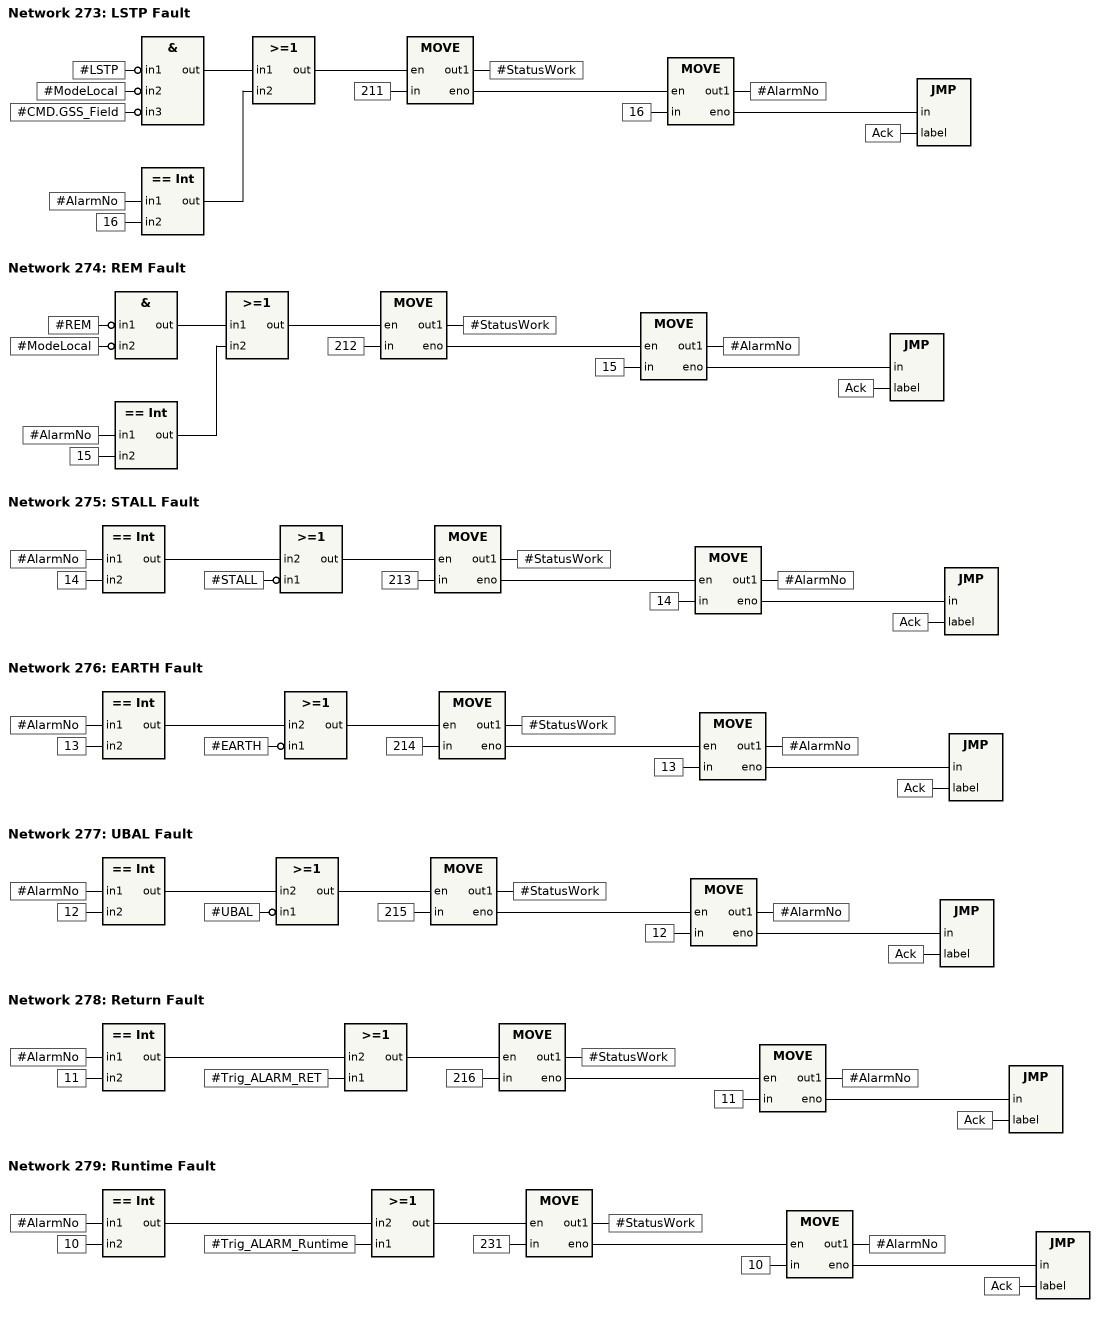
   // ENO of a box is taken as its EN; it also drops when the box reports an error
   #_w1 := (NOT #LSTP AND NOT #ModeLocal AND NOT #CMD.GSS_Field) OR (#AlarmNo = 16);
   IF #_w1 THEN
       #StatusWork := 211;
       #AlarmNo := 16;
       GOTO Ack;
   END_IF;
END_REGION

REGION Network 274: REM Fault
   // ENO of a box is taken as its EN; it also drops when the box reports an error
   #_w1 := (NOT #REM AND NOT #ModeLocal) OR (#AlarmNo = 15);
   IF #_w1 THEN
       #StatusWork := 212;
       #AlarmNo := 15;
       GOTO Ack;
   END_IF;
END_REGION

REGION Network 275: STALL Fault
   // ENO of a box is taken as its EN; it also drops when the box reports an error
   #_w1 := (#AlarmNo = 14) OR NOT #STALL;
   IF #_w1 THEN
       #StatusWork := 213;
       #AlarmNo := 14;
       GOTO Ack;
   END_IF;
END_REGION

REGION Network 276: EARTH Fault
   // ENO of a box is taken as its EN; it also drops when the box reports an error
   #_w1 := (#AlarmNo = 13) OR NOT #EARTH;
   IF #_w1 THEN
       #StatusWork := 214;
       #AlarmNo := 13;
       GOTO Ack;
   END_IF;
END_REGION

REGION Network 277: UBAL Fault
   // ENO of a box is taken as its EN; it also drops when the box reports an error
   #_w1 := (#AlarmNo = 12) OR NOT #UBAL;
   IF #_w1 THEN
       #StatusWork := 215;
       #AlarmNo := 12;
       GOTO Ack;
   END_IF;
END_REGION

REGION Network 278: Return Fault
   // ENO of a box is taken as its EN; it also drops when the box reports an error
   #_w1 := (#AlarmNo = 11) OR #Trig_ALARM_RET;
   IF #_w1 THEN
       #StatusWork := 216;
       #AlarmNo := 11;
       GOTO Ack;
   END_IF;
END_REGION

REGION Network 279: Runtime Fault
   // ENO of a box is taken as its EN; it also drops when the box reports an error
   #_w1 := (#AlarmNo = 10) OR #Trig_ALARM_Runtime;
   IF #_w1 THEN
       #StatusWork := 231;
       #AlarmNo := 10;
       GOTO Ack;
   END_IF;
END_REGION

REGION Network 280: Alarm Switch 1
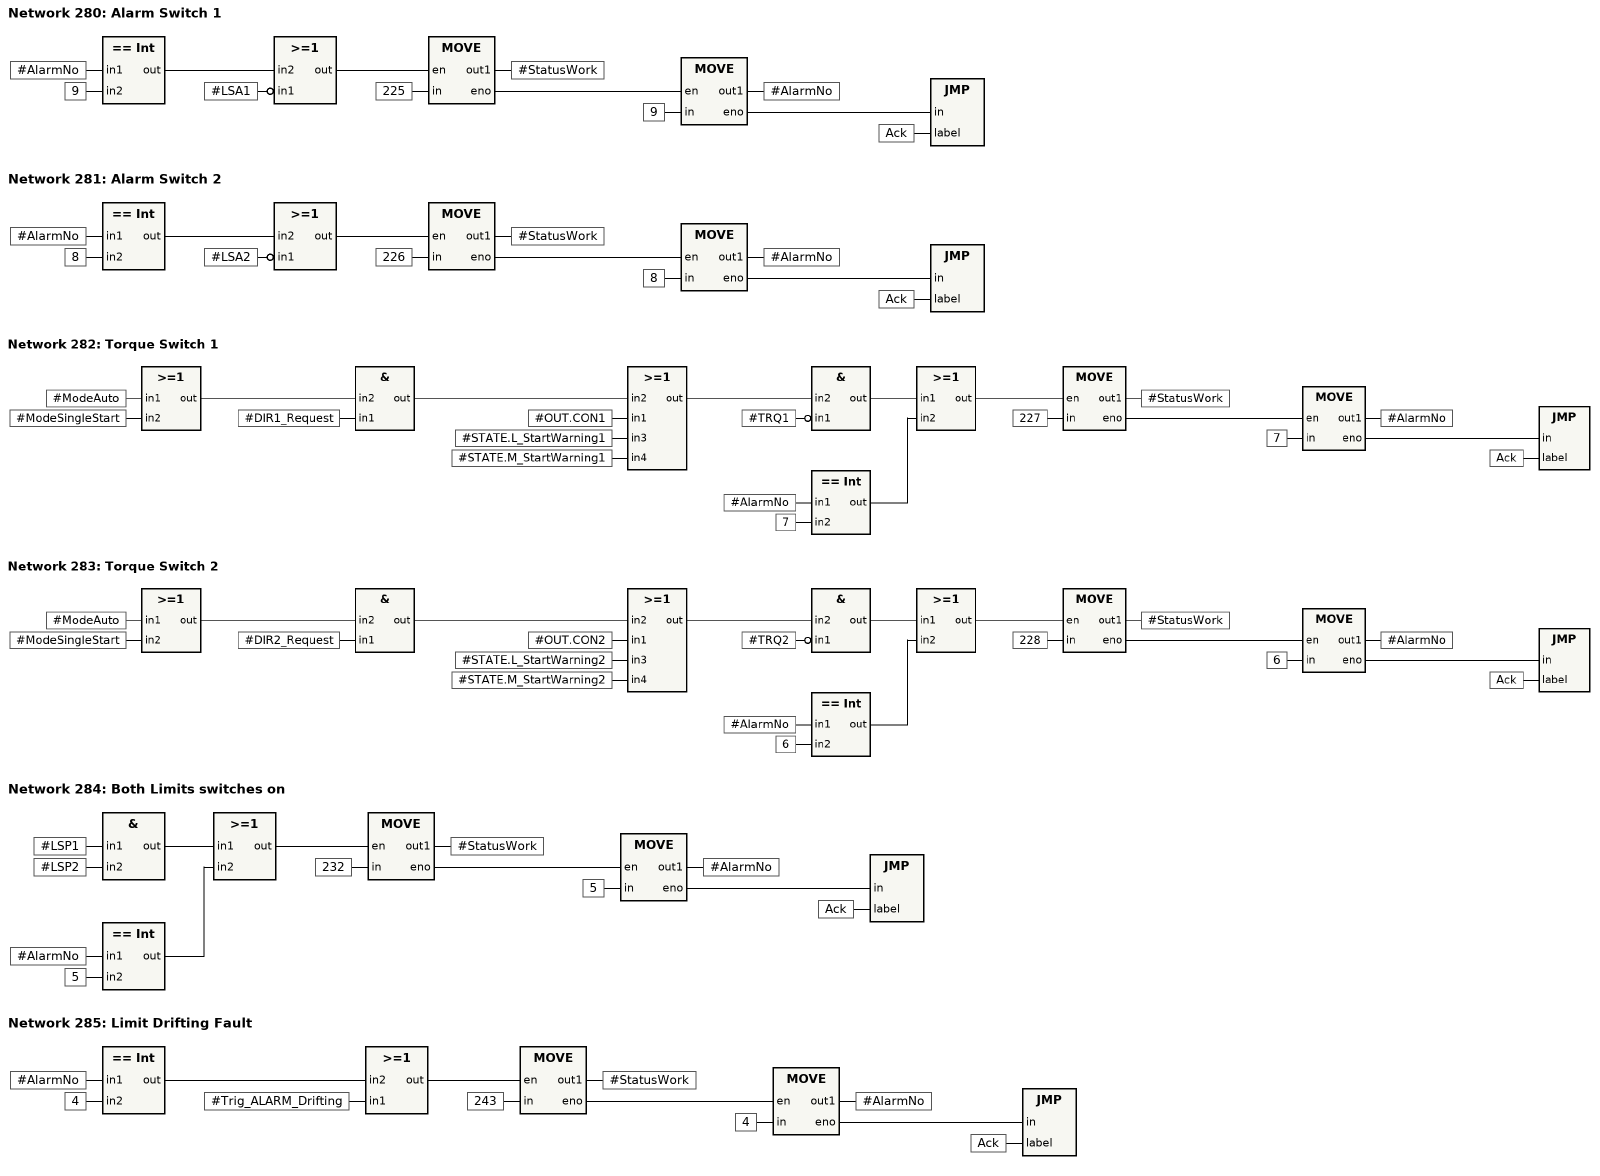
   // ENO of a box is taken as its EN; it also drops when the box reports an error
   #_w1 := (#AlarmNo = 9) OR NOT #LSA1;
   IF #_w1 THEN
       #StatusWork := 225;
       #AlarmNo := 9;
       GOTO Ack;
   END_IF;
END_REGION

REGION Network 281: Alarm Switch 2
   // ENO of a box is taken as its EN; it also drops when the box reports an error
   #_w1 := (#AlarmNo = 8) OR NOT #LSA2;
   IF #_w1 THEN
       #StatusWork := 226;
       #AlarmNo := 8;
       GOTO Ack;
   END_IF;
END_REGION

REGION Network 282: Torque Switch 1
   // Build 006 - 28 Jan 2020 (EXTBOB) : Torque fault considered in Local & Manual start
   // ENO of a box is taken as its EN; it also drops when the box reports an error
   #_w1 := ((((#ModeAuto OR #ModeSingleStart) AND #DIR1_Request) OR #OUT.CON1 OR #STATE.L_StartWarning1 OR #STATE.M_StartWarning1) AND NOT #TRQ1) OR (#AlarmNo = 7);
   IF #_w1 THEN
       #StatusWork := 227;
       #AlarmNo := 7;
       GOTO Ack;
   END_IF;
END_REGION

REGION Network 283: Torque Switch 2
   // Build 006 - 28 Jan 2020 (EXTBOB) : Torque fault considered in Local & Manual start
   // ENO of a box is taken as its EN; it also drops when the box reports an error
   #_w1 := ((((#ModeAuto OR #ModeSingleStart) AND #DIR2_Request) OR #OUT.CON2 OR #STATE.L_StartWarning2 OR #STATE.M_StartWarning2) AND NOT #TRQ2) OR (#AlarmNo = 6);
   IF #_w1 THEN
       #StatusWork := 228;
       #AlarmNo := 6;
       GOTO Ack;
   END_IF;
END_REGION

REGION Network 284: Both Limits switches on
   // ENO of a box is taken as its EN; it also drops when the box reports an error
   #_w1 := (#LSP1 AND #LSP2) OR (#AlarmNo = 5);
   IF #_w1 THEN
       #StatusWork := 232;
       #AlarmNo := 5;
       GOTO Ack;
   END_IF;
END_REGION

REGION Network 285: Limit Drifting Fault
   // ENO of a box is taken as its EN; it also drops when the box reports an error
   #_w1 := (#AlarmNo = 4) OR #Trig_ALARM_Drifting;
   IF #_w1 THEN
       #StatusWork := 243;
       #AlarmNo := 4;
       GOTO Ack;
   END_IF;
END_REGION

REGION Network 286: Analog pos Fault
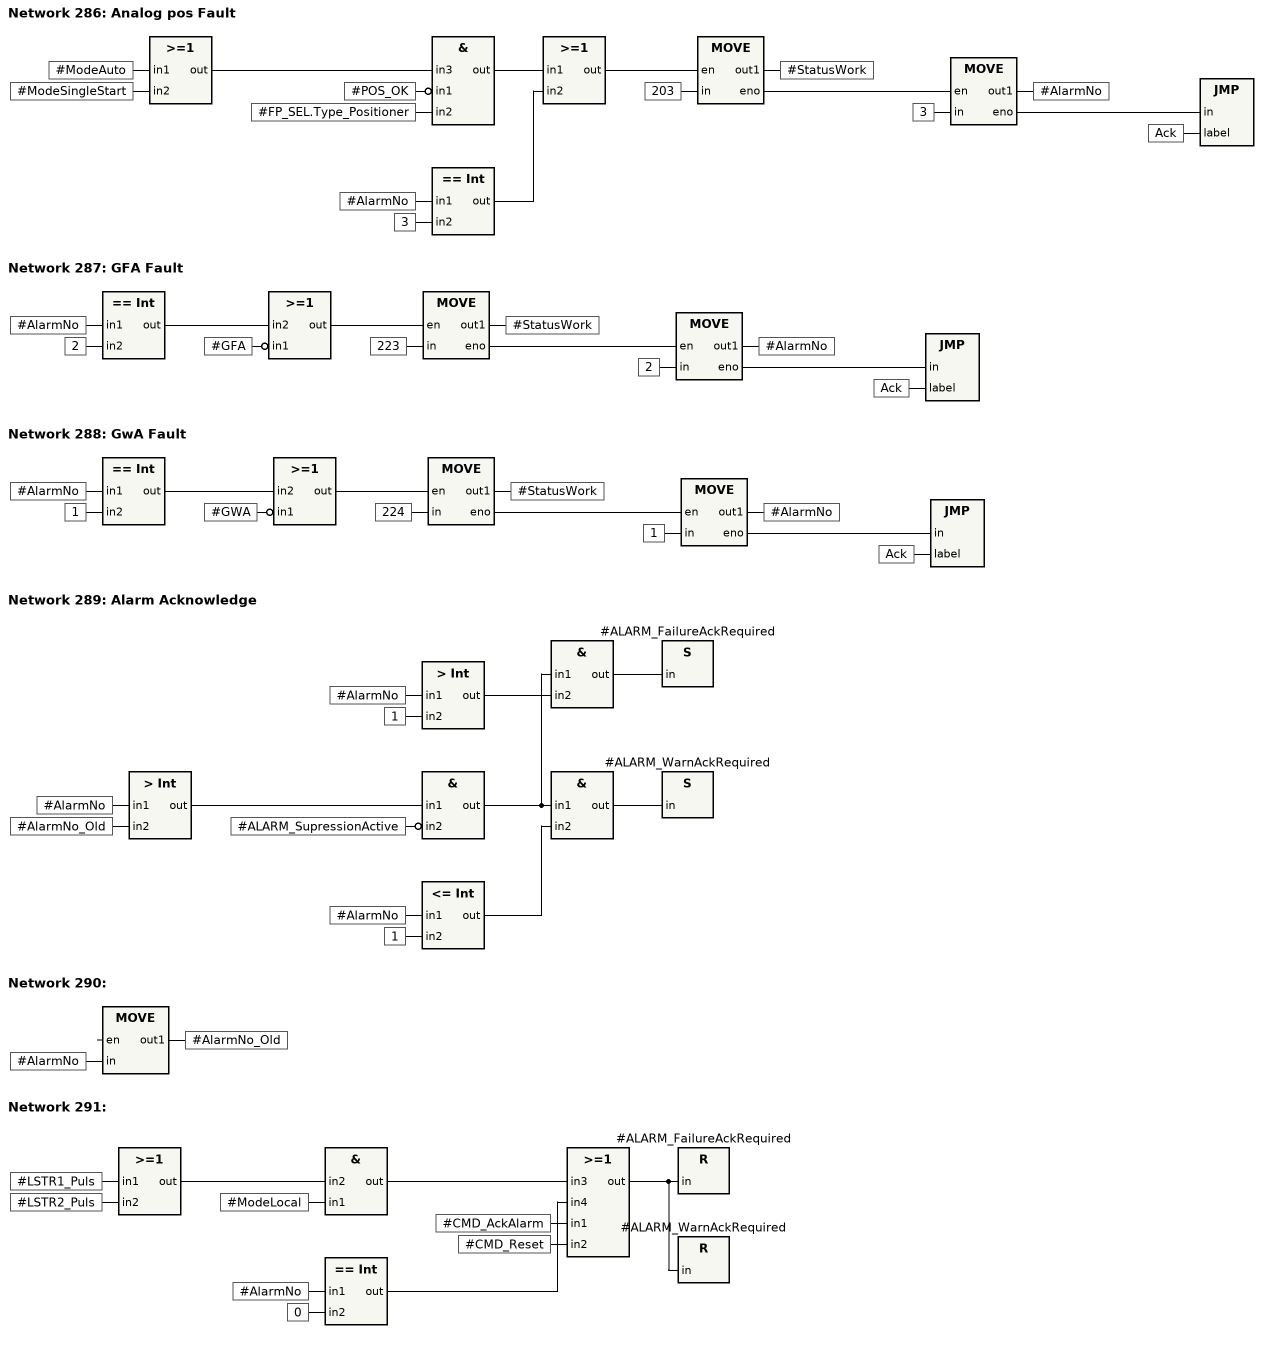
   // ENO of a box is taken as its EN; it also drops when the box reports an error
   #_w1 := ((#ModeAuto OR #ModeSingleStart) AND NOT #POS_OK AND #FP_SEL.Type_Positioner) OR (#AlarmNo = 3);
   IF #_w1 THEN
       #StatusWork := 203;
       #AlarmNo := 3;
       GOTO Ack;
   END_IF;
END_REGION

REGION Network 287: GFA Fault
   // ENO of a box is taken as its EN; it also drops when the box reports an error
   #_w1 := (#AlarmNo = 2) OR NOT #GFA;
   IF #_w1 THEN
       #StatusWork := 223;
       #AlarmNo := 2;
       GOTO Ack;
   END_IF;
END_REGION

REGION Network 288: GwA Fault
   // ENO of a box is taken as its EN; it also drops when the box reports an error
   #_w1 := (#AlarmNo = 1) OR NOT #GWA;
   IF #_w1 THEN
       #StatusWork := 224;
       #AlarmNo := 1;
       GOTO Ack;
   END_IF;
END_REGION

REGION Network 289: Alarm Acknowledge
   Ack:
   #_w1 := (#AlarmNo > #AlarmNo_Old) AND NOT #ALARM_SupressionActive;
   IF #_w1 AND (#AlarmNo > 1) THEN #ALARM_FailureAckRequired := TRUE; END_IF;
   IF #_w1 AND (#AlarmNo <= 1) THEN #ALARM_WarnAckRequired := TRUE; END_IF;
END_REGION

REGION Network 290
   #AlarmNo_Old := #AlarmNo;
END_REGION

REGION Network 291
   IF ((#LSTR1_Puls OR #LSTR2_Puls) AND #ModeLocal) OR (#AlarmNo = 0) OR #CMD_AckAlarm OR #CMD_Reset THEN
       #ALARM_FailureAckRequired := FALSE;
       #ALARM_WarnAckRequired := FALSE;
   END_IF;
END_REGION

REGION Network 292
   // Build 006 - 28 Jan 2020 (EXTBOB) : AlarmNo 6 and 7 Added to prevent Auto ack in torque falut
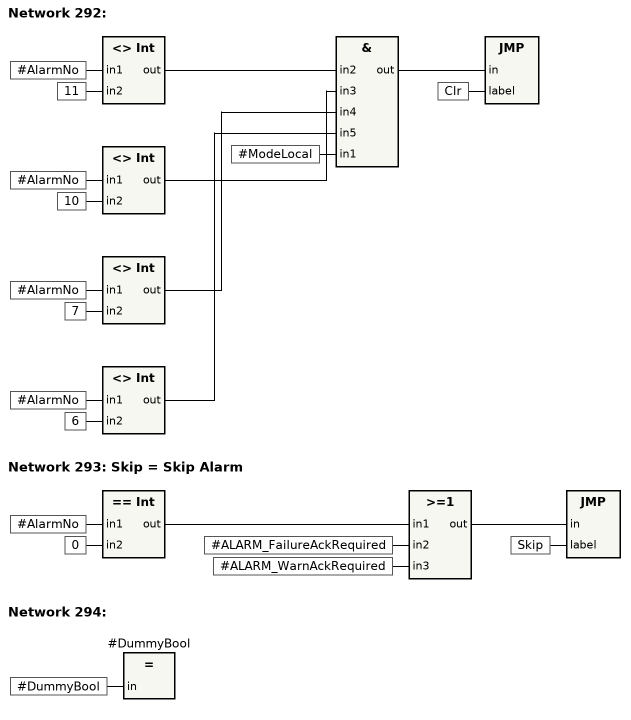
   IF (#AlarmNo <> 11) AND (#AlarmNo <> 10) AND (#AlarmNo <> 7) AND (#AlarmNo <> 6) AND #ModeLocal THEN
       GOTO Clr;
   END_IF;
END_REGION

REGION Network 293: Skip = Skip Alarm
   IF (#AlarmNo = 0) OR #ALARM_FailureAckRequired OR #ALARM_WarnAckRequired THEN GOTO Skip; END_IF;
END_REGION

REGION Network 294
   Clr:
   #DummyBool := #DummyBool;
END_REGION

REGION Network 295
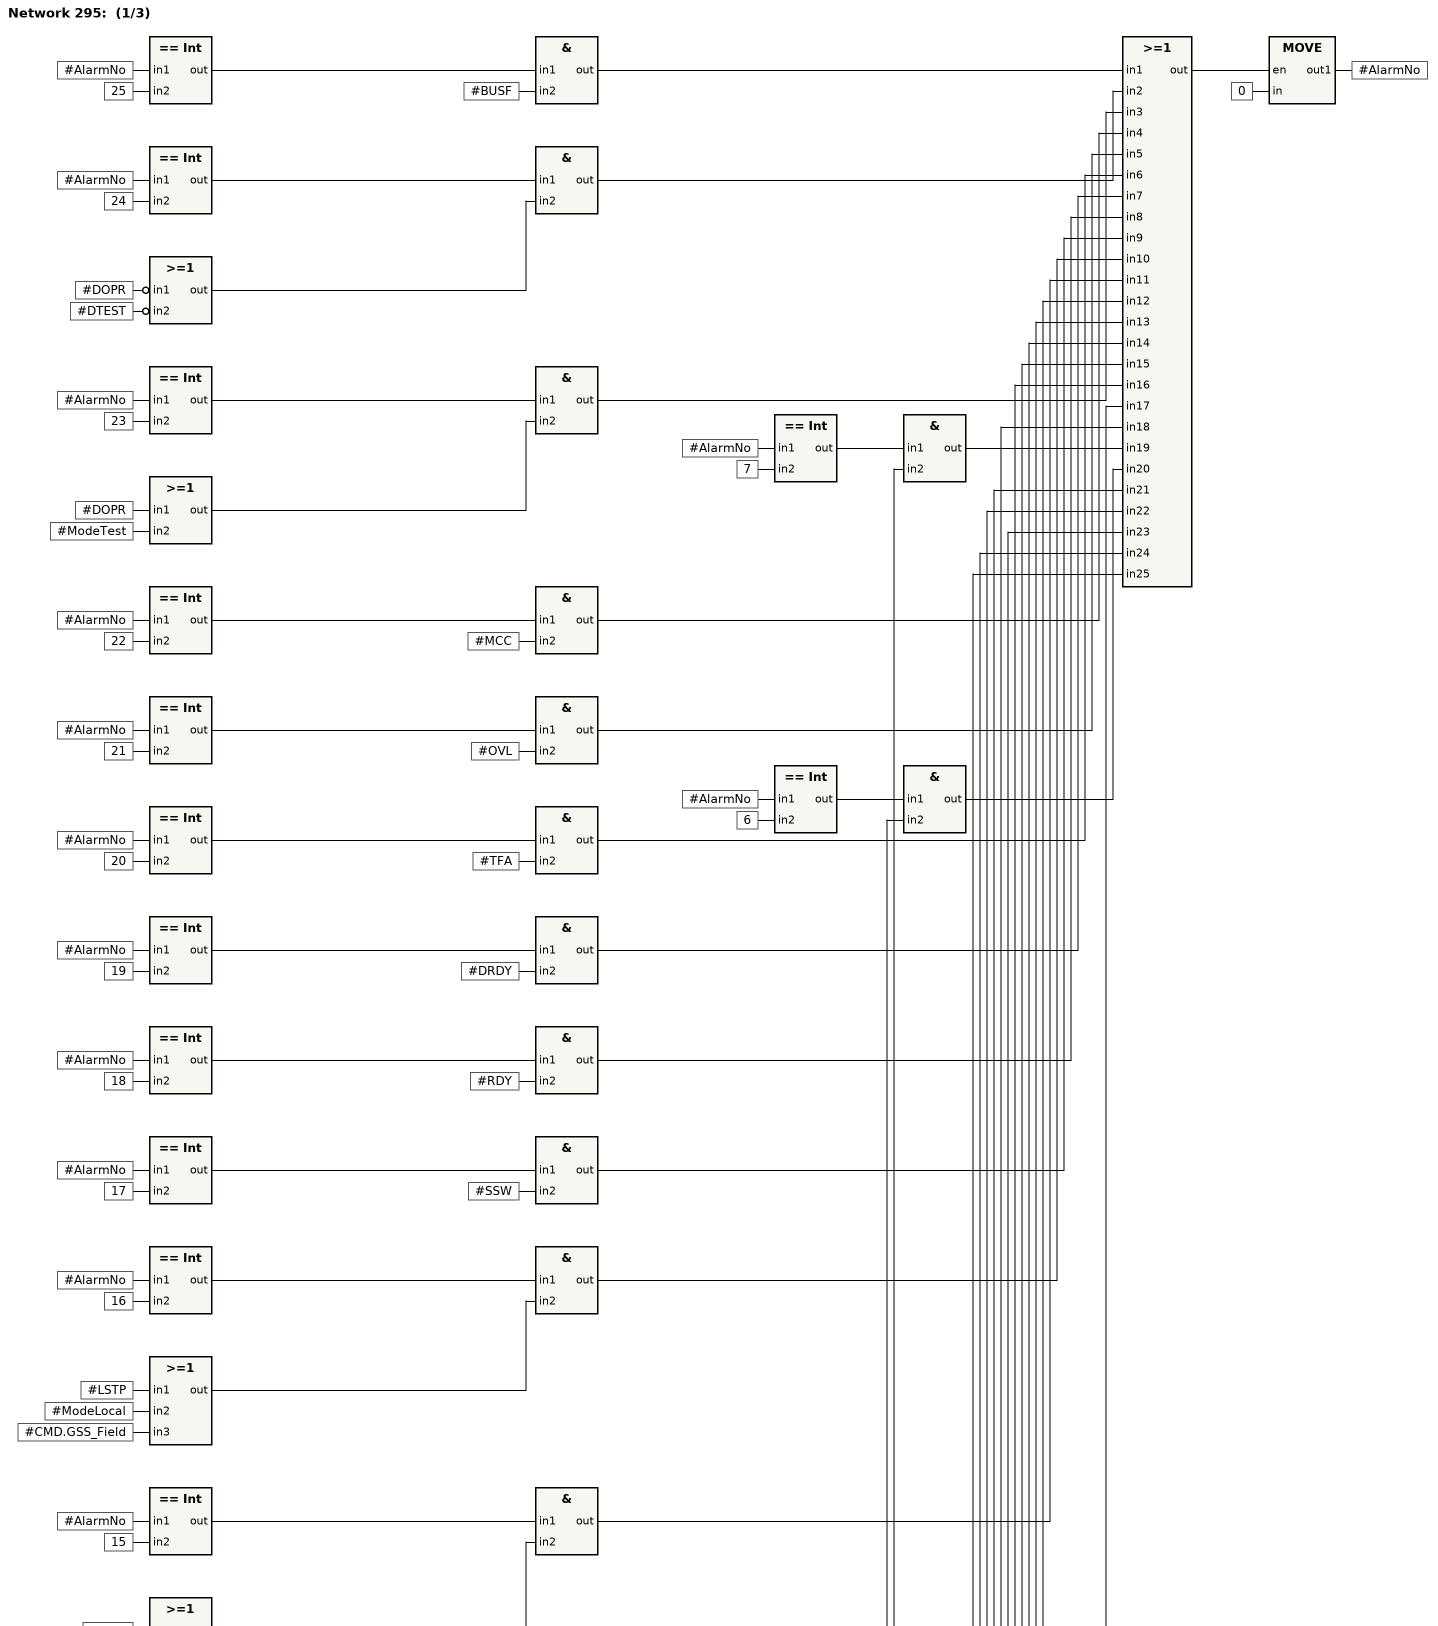
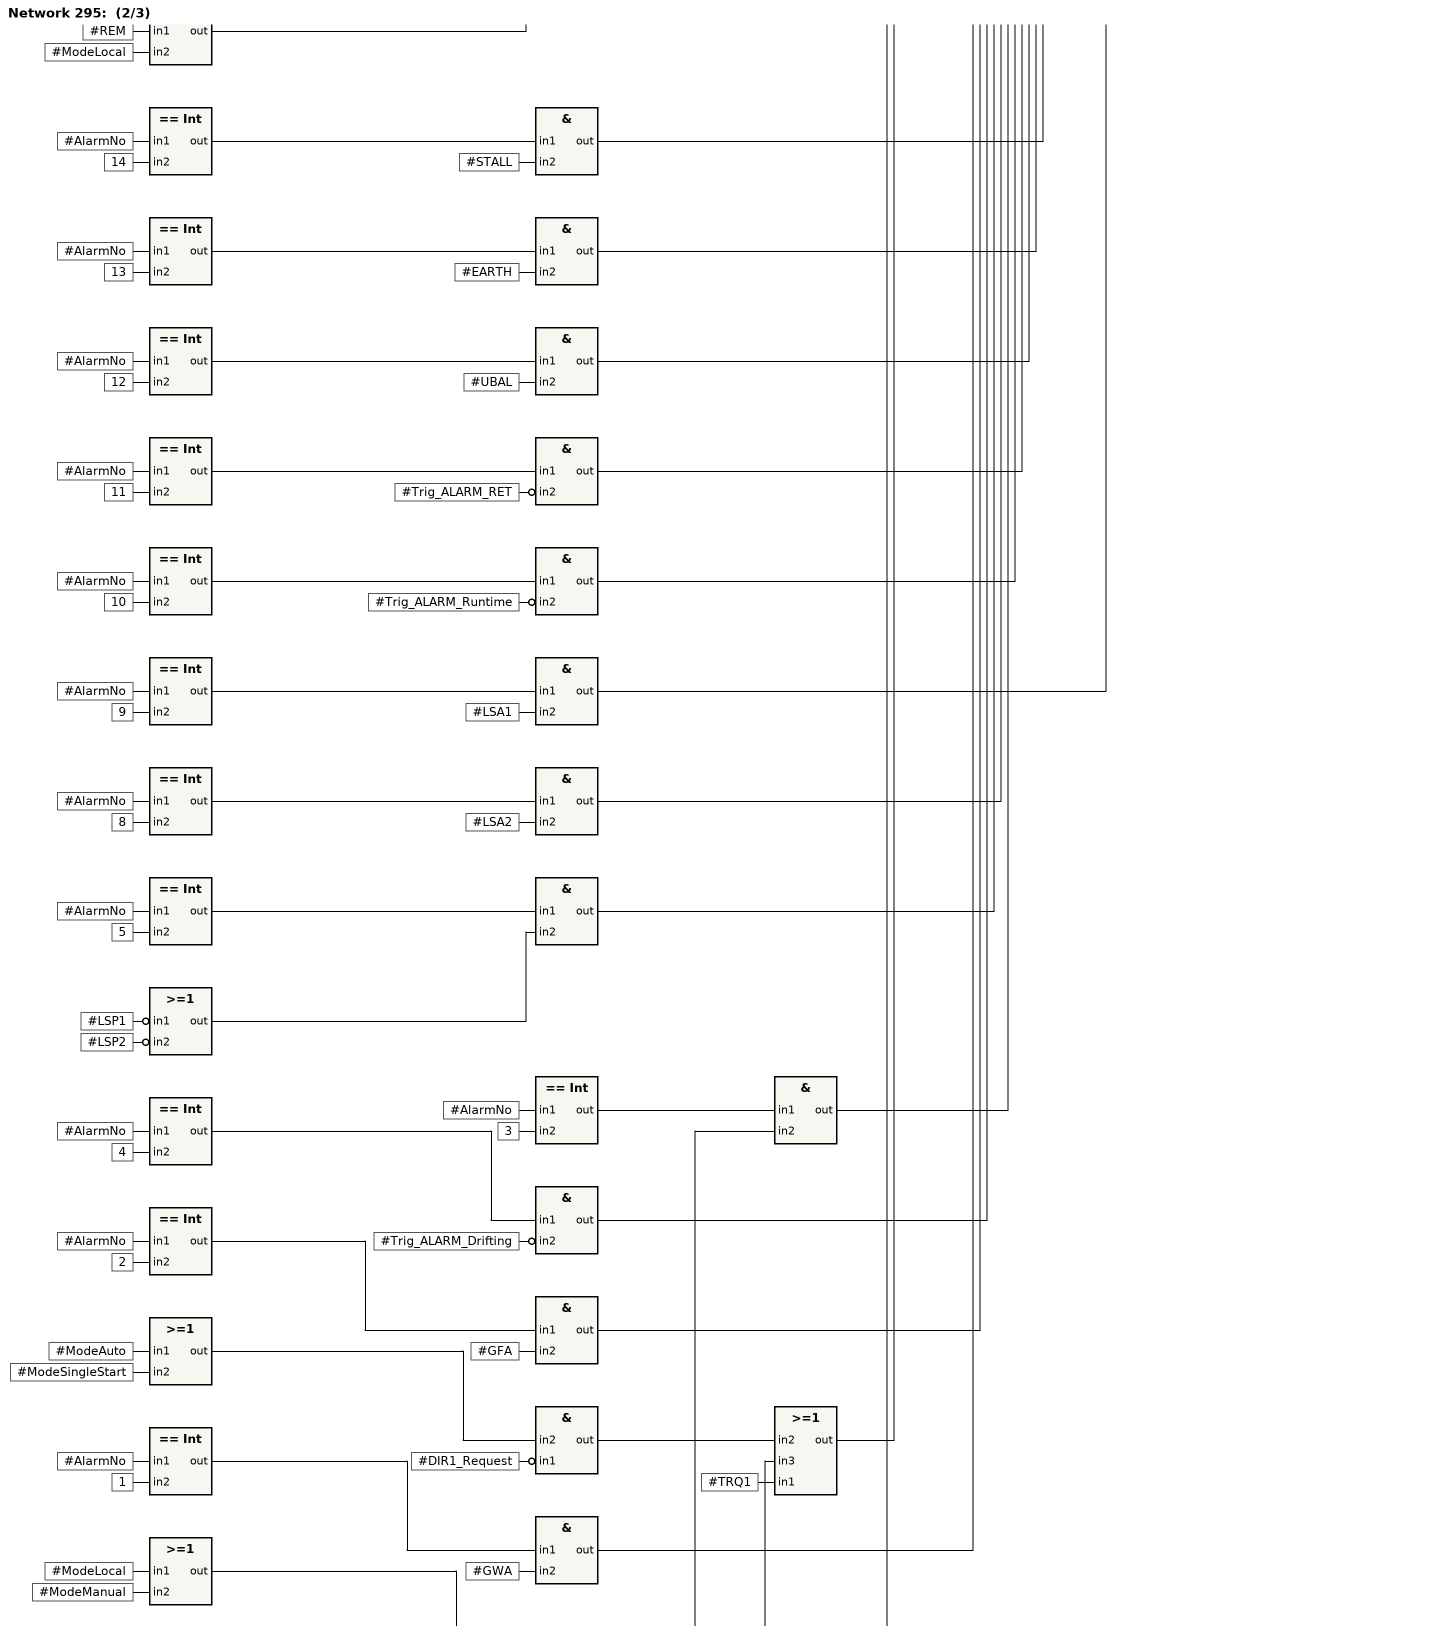
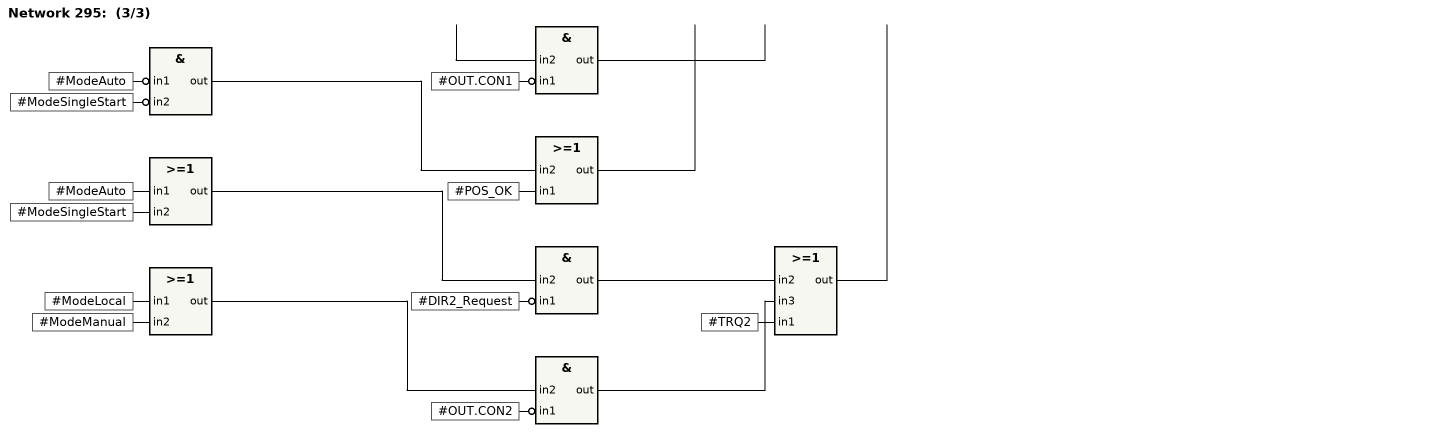
   IF ((#AlarmNo = 25) AND #BUSF) OR ((#AlarmNo = 24) AND (NOT #DOPR OR NOT #DTEST)) OR ((#AlarmNo = 23) AND (#DOPR OR #ModeTest)) OR ((#AlarmNo = 22) AND #MCC) OR ((#AlarmNo = 21) AND #OVL) OR ((#AlarmNo = 20) AND #TFA) OR ((#AlarmNo = 19) AND #DRDY) OR ((#AlarmNo = 18) AND #RDY) OR ((#AlarmNo = 17) AND #SSW) OR ((#AlarmNo = 16) AND (#LSTP OR #ModeLocal OR #CMD.GSS_Field)) OR ((#AlarmNo = 15) AND (#REM OR #ModeLocal)) OR ((#AlarmNo = 14) AND #STALL) OR ((#AlarmNo = 13) AND #EARTH) OR ((#AlarmNo = 12) AND #UBAL) OR ((#AlarmNo = 11) AND NOT #Trig_ALARM_RET) OR ((#AlarmNo = 10) AND NOT #Trig_ALARM_Runtime) OR ((#AlarmNo = 9) AND #LSA1) OR ((#AlarmNo = 8) AND #LSA2) OR ((#AlarmNo = 7) AND (((#ModeAuto OR #ModeSingleStart) AND NOT #DIR1_Request) OR ((#ModeLocal OR #ModeManual) AND NOT #OUT.CON1) OR #TRQ1)) OR ((#AlarmNo = 6) AND (((#ModeAuto OR #ModeSingleStart) AND NOT #DIR2_Request) OR ((#ModeLocal OR #ModeManual) AND NOT #OUT.CON2) OR #TRQ2)) OR ((#AlarmNo = 5) AND (NOT #LSP1 OR NOT #LSP2)) OR ((#AlarmNo = 4) AND NOT #Trig_ALARM_Drifting) OR ((#AlarmNo = 3) AND ((NOT #ModeAuto AND NOT #ModeSingleStart) OR #POS_OK)) OR ((#AlarmNo = 2) AND #GFA) OR ((#AlarmNo = 1) AND #GWA) THEN
       #AlarmNo := 0;
   END_IF;
END_REGION

REGION Network 296
   // Build 006 - 28 Jan 2020 (EXTBOB) : Newly added to make this logic same as other PLC brands, it will overcome the not generation of alarm in local mode wrt local start pulse, alarm ack req set/reset in one scan
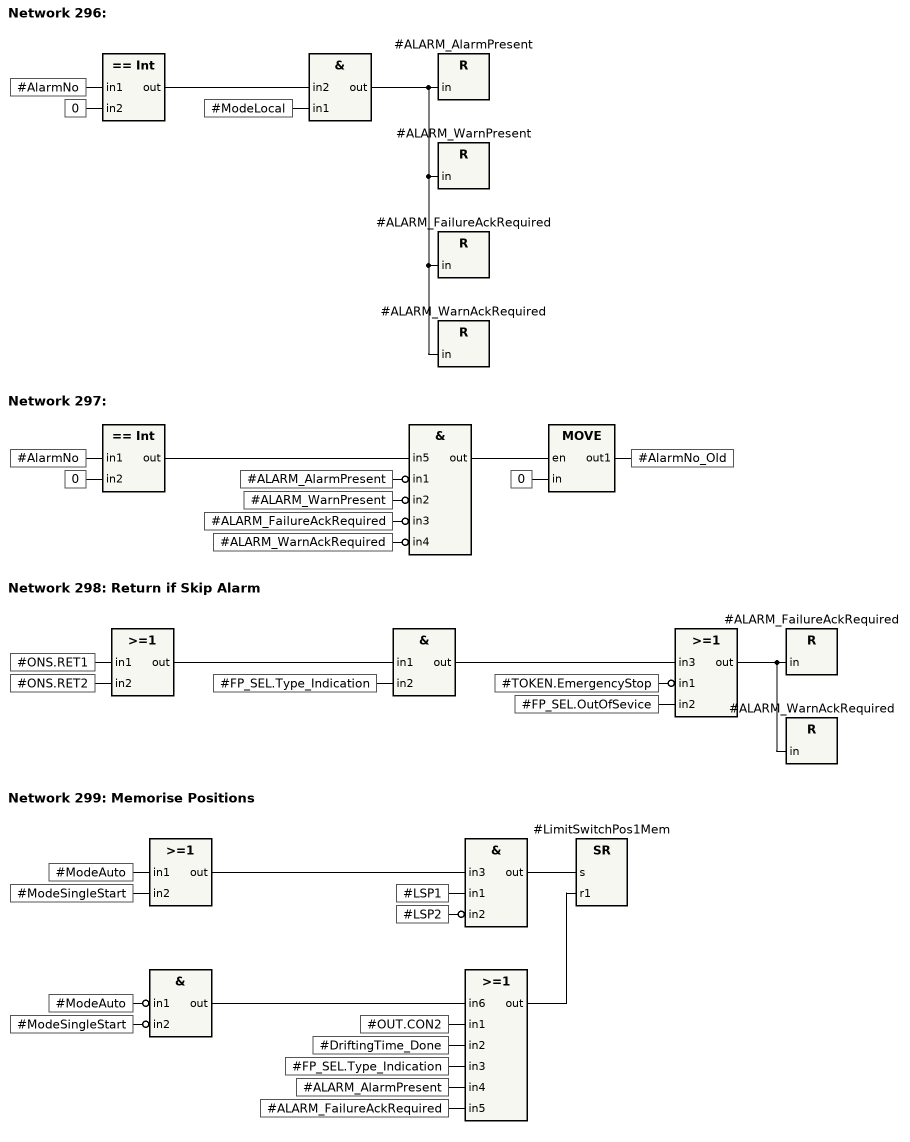
   IF (#AlarmNo = 0) AND #ModeLocal THEN
       #ALARM_AlarmPresent := FALSE;
       #ALARM_WarnPresent := FALSE;
       #ALARM_FailureAckRequired := FALSE;
       #ALARM_WarnAckRequired := FALSE;
   END_IF;
END_REGION

REGION Network 297
   IF (#AlarmNo = 0) AND NOT #ALARM_AlarmPresent AND NOT #ALARM_WarnPresent AND NOT #ALARM_FailureAckRequired AND NOT #ALARM_WarnAckRequired THEN
       #AlarmNo_Old := 0;
   END_IF;
END_REGION

REGION Network 298: Return if Skip Alarm
   // Build 002: 26 March 2019 : Alarm/Warning are Auto Acknowledged on OutOfService
   // Build 003 - 30 June 2019 (EXTBOB) : Acknowledge pending alarms when Unit started as "Indication"
   Skip:
   IF ((#ONS.RET1 OR #ONS.RET2) AND #FP_SEL.Type_Indication) OR NOT #TOKEN.EmergencyStop OR #FP_SEL.OutOfSevice THEN
       #ALARM_FailureAckRequired := FALSE;
       #ALARM_WarnAckRequired := FALSE;
   END_IF;
END_REGION

REGION Network 299: Memorise Positions
   // Build 005 - 24 Oct 2019 : Alarm Present & Aalrm failure Ack flag are added to prevent limit driftinmg during an alarm
   IF (#ModeAuto OR #ModeSingleStart) AND #LSP1 AND NOT #LSP2 THEN
       #LimitSwitchPos1Mem := TRUE;   // SR flip-flop
   END_IF;
   IF (NOT #ModeAuto AND NOT #ModeSingleStart) OR #OUT.CON2 OR #DriftingTime_Done OR #FP_SEL.Type_Indication OR #ALARM_AlarmPresent OR #ALARM_FailureAckRequired THEN
       #LimitSwitchPos1Mem := FALSE;
   END_IF;
END_REGION

REGION Network 300
   // Build 005 - 24 Oct 2019 : Alarm Present & Aalrm failure Ack flag are added to prevent limit driftinmg during an alarm
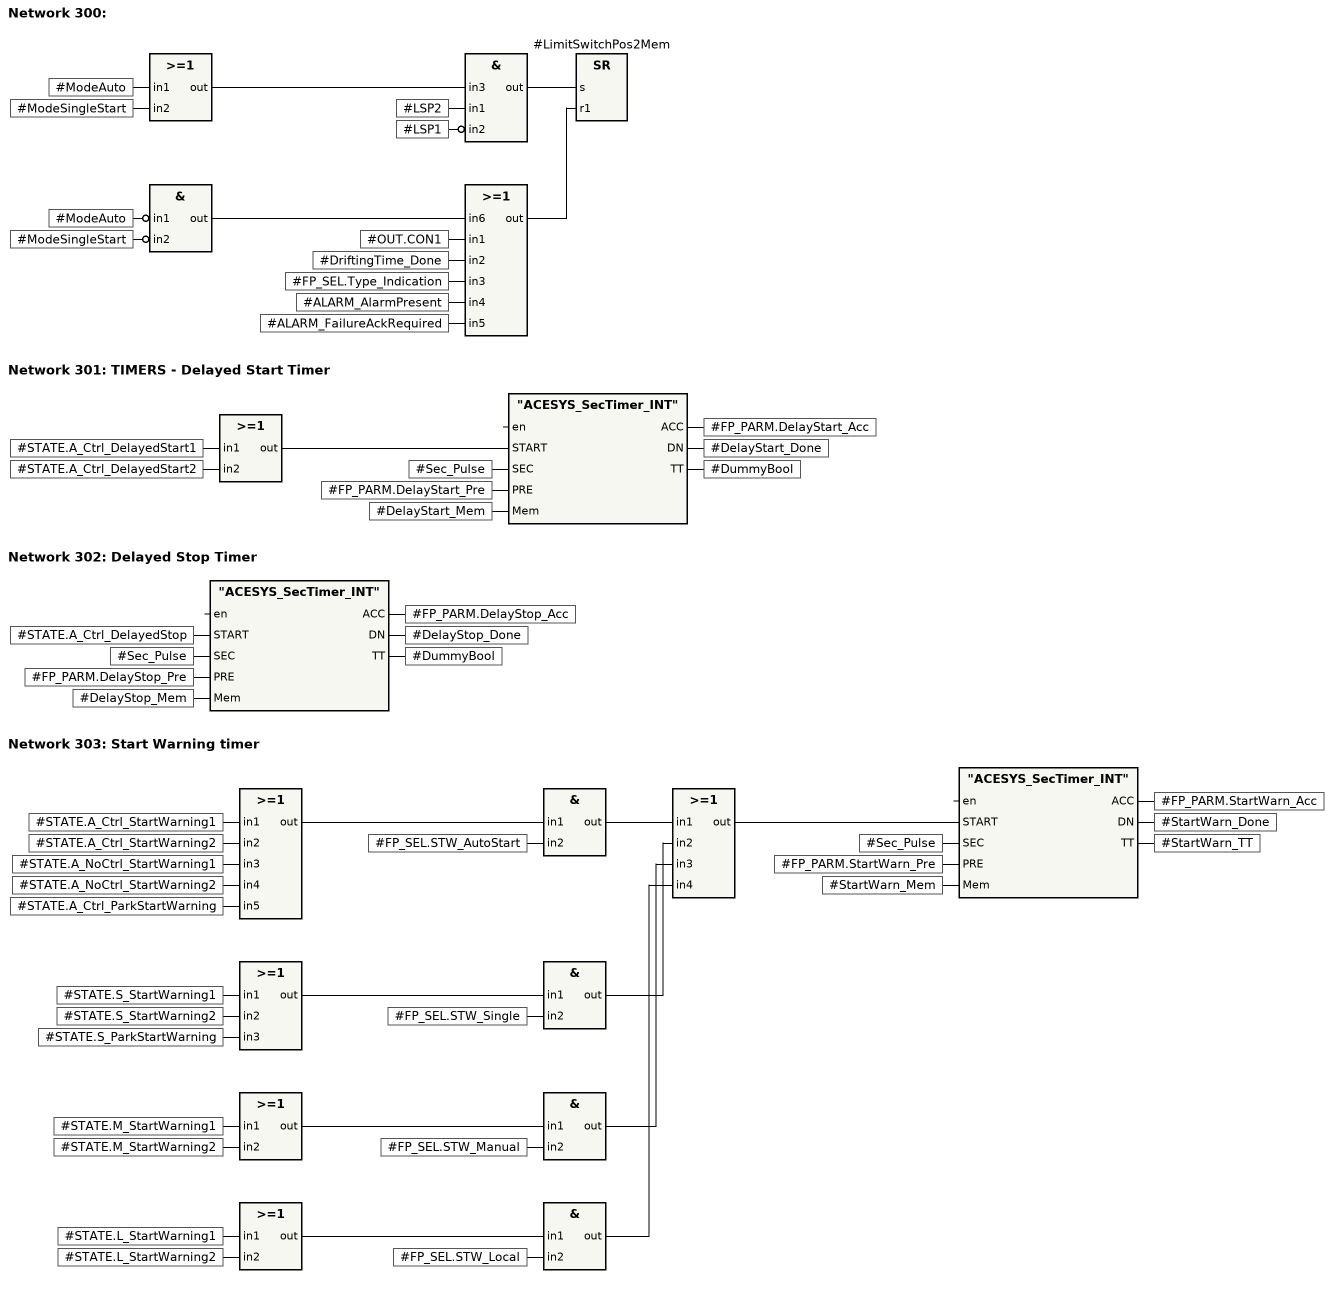
   IF (#ModeAuto OR #ModeSingleStart) AND #LSP2 AND NOT #LSP1 THEN
       #LimitSwitchPos2Mem := TRUE;   // SR flip-flop
   END_IF;
   IF (NOT #ModeAuto AND NOT #ModeSingleStart) OR #OUT.CON1 OR #DriftingTime_Done OR #FP_SEL.Type_Indication OR #ALARM_AlarmPresent OR #ALARM_FailureAckRequired THEN
       #LimitSwitchPos2Mem := FALSE;
   END_IF;
END_REGION

REGION Network 301: TIMERS - Delayed Start Timer
   "ACESYS_SecTimer_INT"(START := #STATE.A_Ctrl_DelayedStart1 OR #STATE.A_Ctrl_DelayedStart2,
                         SEC := #Sec_Pulse,
                         PRE := #FP_PARM.DelayStart_Pre,
                         Mem := #DelayStart_Mem,
                         ACC => #FP_PARM.DelayStart_Acc,
                         DN => #DelayStart_Done,
                         TT => #DummyBool);
END_REGION

REGION Network 302: Delayed Stop Timer
   "ACESYS_SecTimer_INT"(START := #STATE.A_Ctrl_DelayedStop,
                         SEC := #Sec_Pulse,
                         PRE := #FP_PARM.DelayStop_Pre,
                         Mem := #DelayStop_Mem,
                         ACC => #FP_PARM.DelayStop_Acc,
                         DN => #DelayStop_Done,
                         TT => #DummyBool);
END_REGION

REGION Network 303: Start Warning timer
   "ACESYS_SecTimer_INT"(START := ((#STATE.A_Ctrl_StartWarning1 OR #STATE.A_Ctrl_StartWarning2 OR #STATE.A_NoCtrl_StartWarning1 OR #STATE.A_NoCtrl_StartWarning2 OR #STATE.A_Ctrl_ParkStartWarning) AND #FP_SEL.STW_AutoStart) OR ((#STATE.S_StartWarning1 OR #STATE.S_StartWarning2 OR #STATE.S_ParkStartWarning) AND #FP_SEL.STW_Single) OR ((#STATE.M_StartWarning1 OR #STATE.M_StartWarning2) AND #FP_SEL.STW_Manual) OR ((#STATE.L_StartWarning1 OR #STATE.L_StartWarning2) AND #FP_SEL.STW_Local),
                         SEC := #Sec_Pulse,
                         PRE := #FP_PARM.StartWarn_Pre,
                         Mem := #StartWarn_Mem,
                         ACC => #FP_PARM.StartWarn_Acc,
                         DN => #StartWarn_Done,
                         TT => #StartWarn_TT);
END_REGION

REGION Network 304: Direction Change Timers
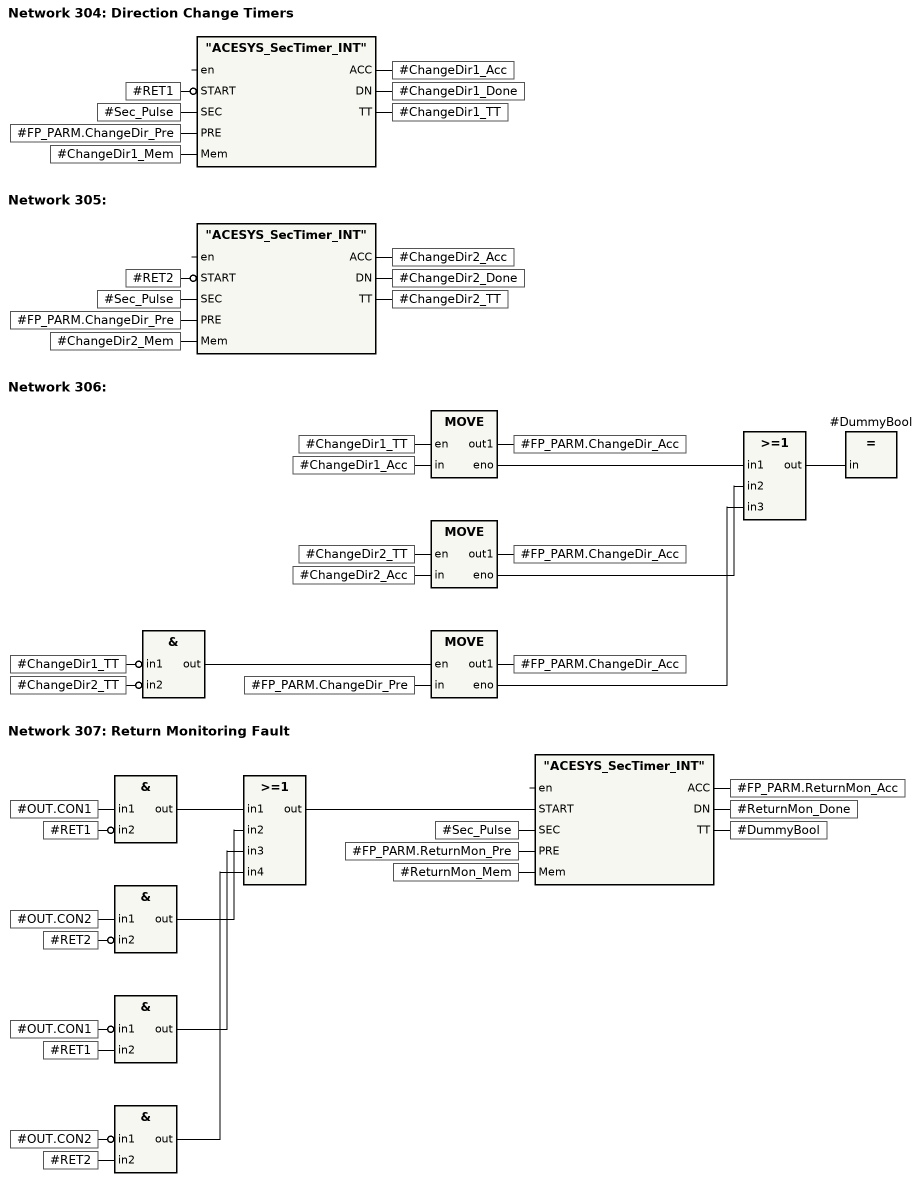
   "ACESYS_SecTimer_INT"(START := NOT #RET1,
                         SEC := #Sec_Pulse,
                         PRE := #FP_PARM.ChangeDir_Pre,
                         Mem := #ChangeDir1_Mem,
                         ACC => #ChangeDir1_Acc,
                         DN => #ChangeDir1_Done,
                         TT => #ChangeDir1_TT);
END_REGION

REGION Network 305
   "ACESYS_SecTimer_INT"(START := NOT #RET2,
                         SEC := #Sec_Pulse,
                         PRE := #FP_PARM.ChangeDir_Pre,
                         Mem := #ChangeDir2_Mem,
                         ACC => #ChangeDir2_Acc,
                         DN => #ChangeDir2_Done,
                         TT => #ChangeDir2_TT);
END_REGION

REGION Network 306
   // ENO of a box is taken as its EN; it also drops when the box reports an error
   IF #ChangeDir1_TT THEN #FP_PARM.ChangeDir_Acc := #ChangeDir1_Acc; END_IF;
   IF #ChangeDir2_TT THEN #FP_PARM.ChangeDir_Acc := #ChangeDir2_Acc; END_IF;
   #_w1 := NOT #ChangeDir1_TT AND NOT #ChangeDir2_TT;
   IF #_w1 THEN #FP_PARM.ChangeDir_Acc := #FP_PARM.ChangeDir_Pre; END_IF;
   #DummyBool := #ChangeDir1_TT OR #ChangeDir2_TT OR #_w1;
END_REGION

REGION Network 307: Return Monitoring Fault
   "ACESYS_SecTimer_INT"(START := (#OUT.CON1 AND NOT #RET1) OR (#OUT.CON2 AND NOT #RET2) OR (NOT #OUT.CON1 AND #RET1) OR (NOT #OUT.CON2 AND #RET2),
                         SEC := #Sec_Pulse,
                         PRE := #FP_PARM.ReturnMon_Pre,
                         Mem := #ReturnMon_Mem,
                         ACC => #FP_PARM.ReturnMon_Acc,
                         DN => #ReturnMon_Done,
                         TT => #DummyBool);
END_REGION

REGION Network 308
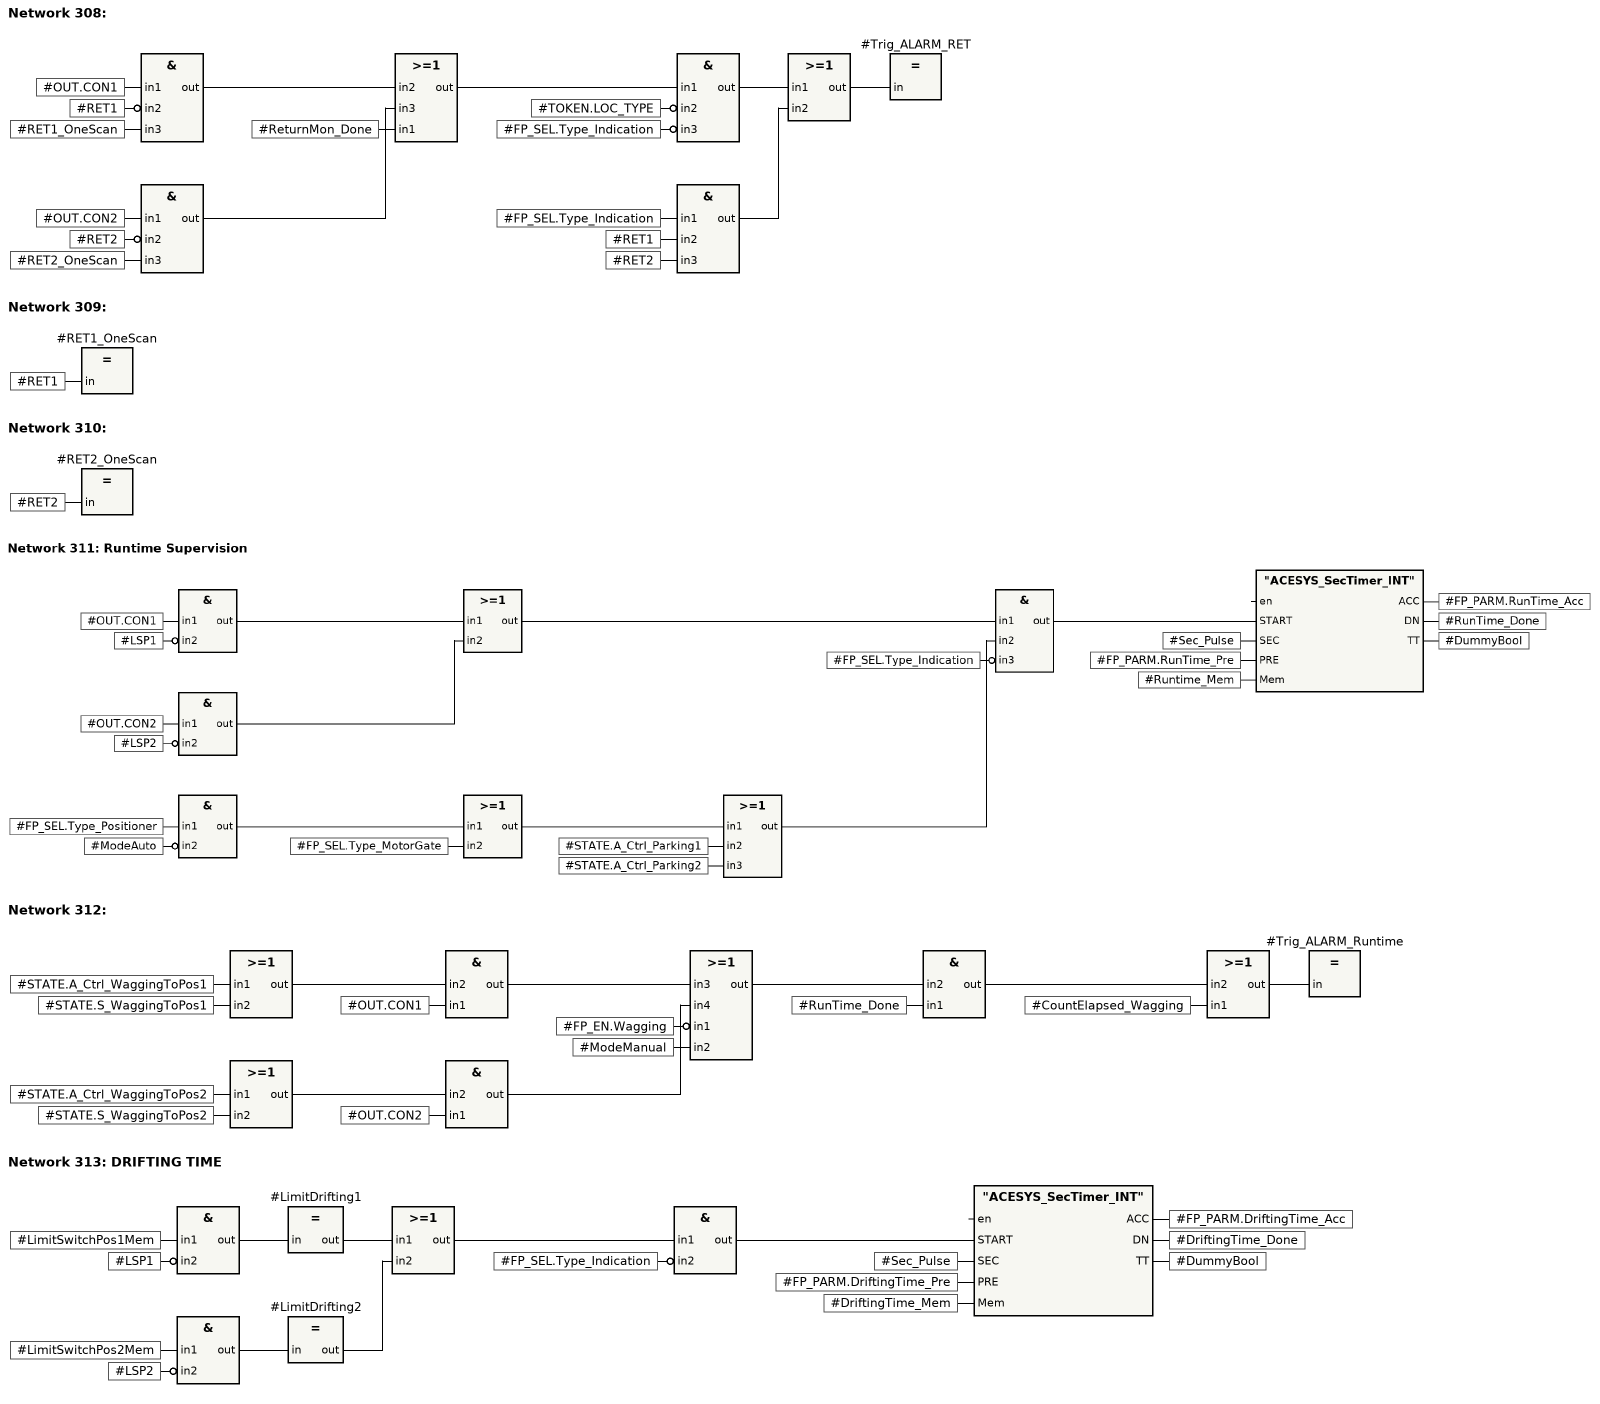
   #Trig_ALARM_RET := (((#OUT.CON1 AND NOT #RET1 AND #RET1_OneScan) OR (#OUT.CON2 AND NOT #RET2 AND #RET2_OneScan) OR #ReturnMon_Done) AND NOT #TOKEN.LOC_TYPE AND NOT #FP_SEL.Type_Indication) OR (#FP_SEL.Type_Indication AND #RET1 AND #RET2);
END_REGION

REGION Network 309
   #RET1_OneScan := #RET1;
END_REGION

REGION Network 310
   #RET2_OneScan := #RET2;
END_REGION

REGION Network 311: Runtime Supervision
   "ACESYS_SecTimer_INT"(START := ((#OUT.CON1 AND NOT #LSP1) OR (#OUT.CON2 AND NOT #LSP2)) AND ((#FP_SEL.Type_Positioner AND NOT #ModeAuto) OR #FP_SEL.Type_MotorGate OR #STATE.A_Ctrl_Parking1 OR #STATE.A_Ctrl_Parking2) AND NOT #FP_SEL.Type_Indication,
                         SEC := #Sec_Pulse,
                         PRE := #FP_PARM.RunTime_Pre,
                         Mem := #Runtime_Mem,
                         ACC => #FP_PARM.RunTime_Acc,
                         DN => #RunTime_Done,
                         TT => #DummyBool);
END_REGION

REGION Network 312
   #Trig_ALARM_Runtime := ((((#STATE.A_Ctrl_WaggingToPos1 OR #STATE.S_WaggingToPos1) AND #OUT.CON1) OR ((#STATE.A_Ctrl_WaggingToPos2 OR #STATE.S_WaggingToPos2) AND #OUT.CON2) OR NOT #FP_EN.Wagging OR #ModeManual) AND #RunTime_Done) OR #CountElapsed_Wagging;
END_REGION

REGION Network 313: DRIFTING TIME
   #LimitDrifting1 := #LimitSwitchPos1Mem AND NOT #LSP1;
   #LimitDrifting2 := #LimitSwitchPos2Mem AND NOT #LSP2;
   "ACESYS_SecTimer_INT"(START := (#LimitDrifting1 OR #LimitDrifting2) AND NOT #FP_SEL.Type_Indication,
                         SEC := #Sec_Pulse,
                         PRE := #FP_PARM.DriftingTime_Pre,
                         Mem := #DriftingTime_Mem,
                         ACC => #FP_PARM.DriftingTime_Acc,
                         DN => #DriftingTime_Done,
                         TT => #DummyBool);
END_REGION

REGION Network 314
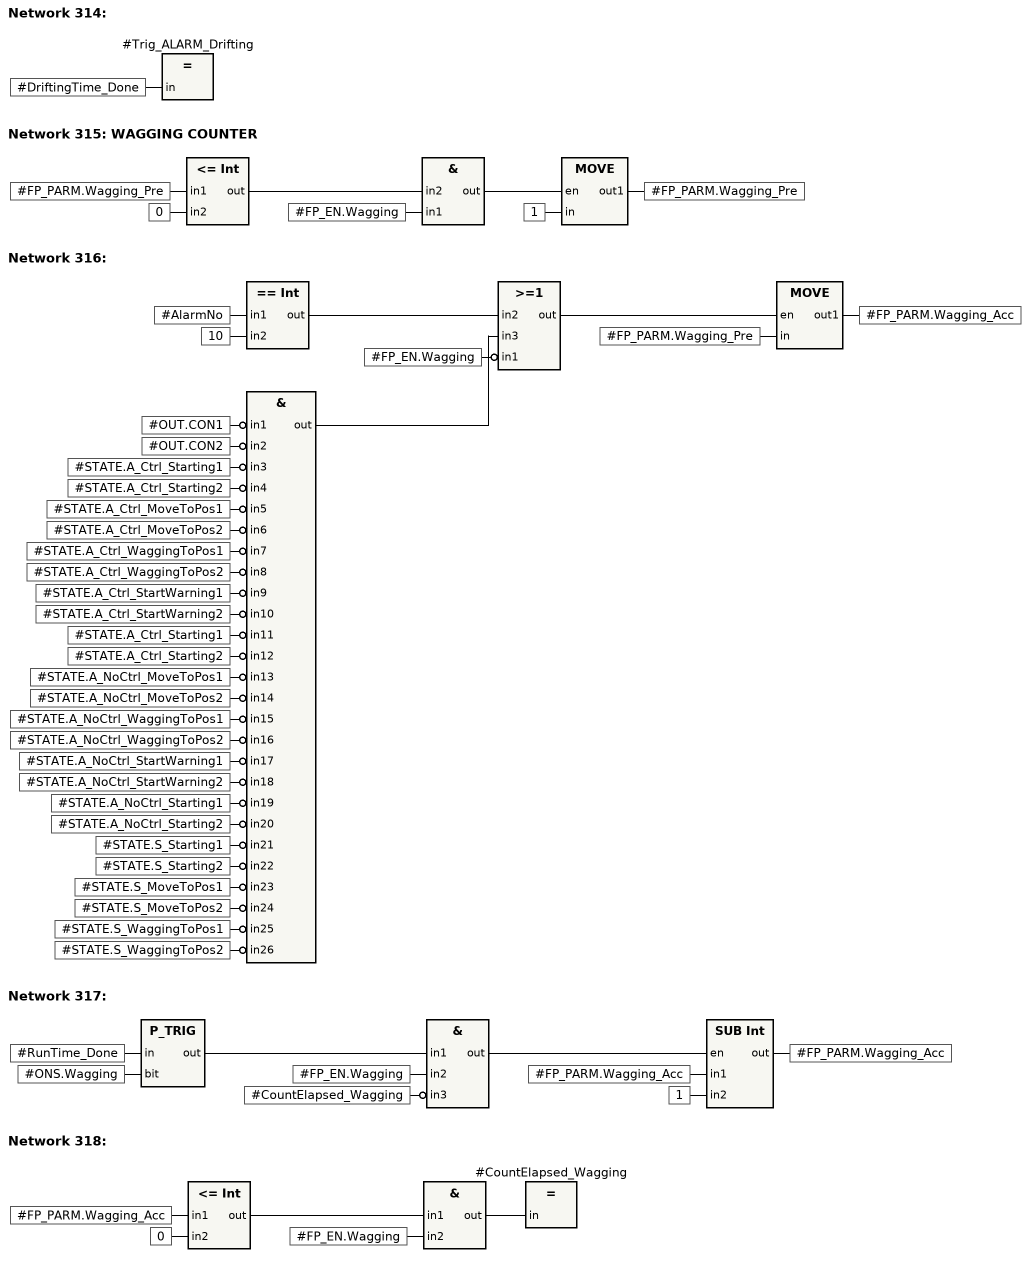
   #Trig_ALARM_Drifting := #DriftingTime_Done;
END_REGION

REGION Network 315: WAGGING COUNTER
   IF (#FP_PARM.Wagging_Pre <= 0) AND #FP_EN.Wagging THEN #FP_PARM.Wagging_Pre := 1; END_IF;
END_REGION

REGION Network 316
   IF (#AlarmNo = 10) OR (NOT #OUT.CON1 AND NOT #OUT.CON2 AND NOT #STATE.A_Ctrl_Starting1 AND NOT #STATE.A_Ctrl_Starting2 AND NOT #STATE.A_Ctrl_MoveToPos1 AND NOT #STATE.A_Ctrl_MoveToPos2 AND NOT #STATE.A_Ctrl_WaggingToPos1 AND NOT #STATE.A_Ctrl_WaggingToPos2 AND NOT #STATE.A_Ctrl_StartWarning1 AND NOT #STATE.A_Ctrl_StartWarning2 AND NOT #STATE.A_Ctrl_Starting1 AND NOT #STATE.A_Ctrl_Starting2 AND NOT #STATE.A_NoCtrl_MoveToPos1 AND NOT #STATE.A_NoCtrl_MoveToPos2 AND NOT #STATE.A_NoCtrl_WaggingToPos1 AND NOT #STATE.A_NoCtrl_WaggingToPos2 AND NOT #STATE.A_NoCtrl_StartWarning1 AND NOT #STATE.A_NoCtrl_StartWarning2 AND NOT #STATE.A_NoCtrl_Starting1 AND NOT #STATE.A_NoCtrl_Starting2 AND NOT #STATE.S_Starting1 AND NOT #STATE.S_Starting2 AND NOT #STATE.S_MoveToPos1 AND NOT #STATE.S_MoveToPos2 AND NOT #STATE.S_WaggingToPos1 AND NOT #STATE.S_WaggingToPos2) OR NOT #FP_EN.Wagging THEN
       #FP_PARM.Wagging_Acc := #FP_PARM.Wagging_Pre;
   END_IF;
END_REGION

REGION Network 317
   #_w1 := #RunTime_Done AND NOT #ONS.Wagging;   // rising edge
   #ONS.Wagging := #RunTime_Done;
   IF #_w1 AND #FP_EN.Wagging AND NOT #CountElapsed_Wagging THEN
       #FP_PARM.Wagging_Acc := #FP_PARM.Wagging_Acc - 1;
   END_IF;
END_REGION

REGION Network 318
   #CountElapsed_Wagging := (#FP_PARM.Wagging_Acc <= 0) AND #FP_EN.Wagging;
END_REGION

REGION Network 319: OUTPUTS
   // Build 003 - 2.July.2019 (EXTBOB): Added LOC_TYPE to prevent output being energized when running from the field
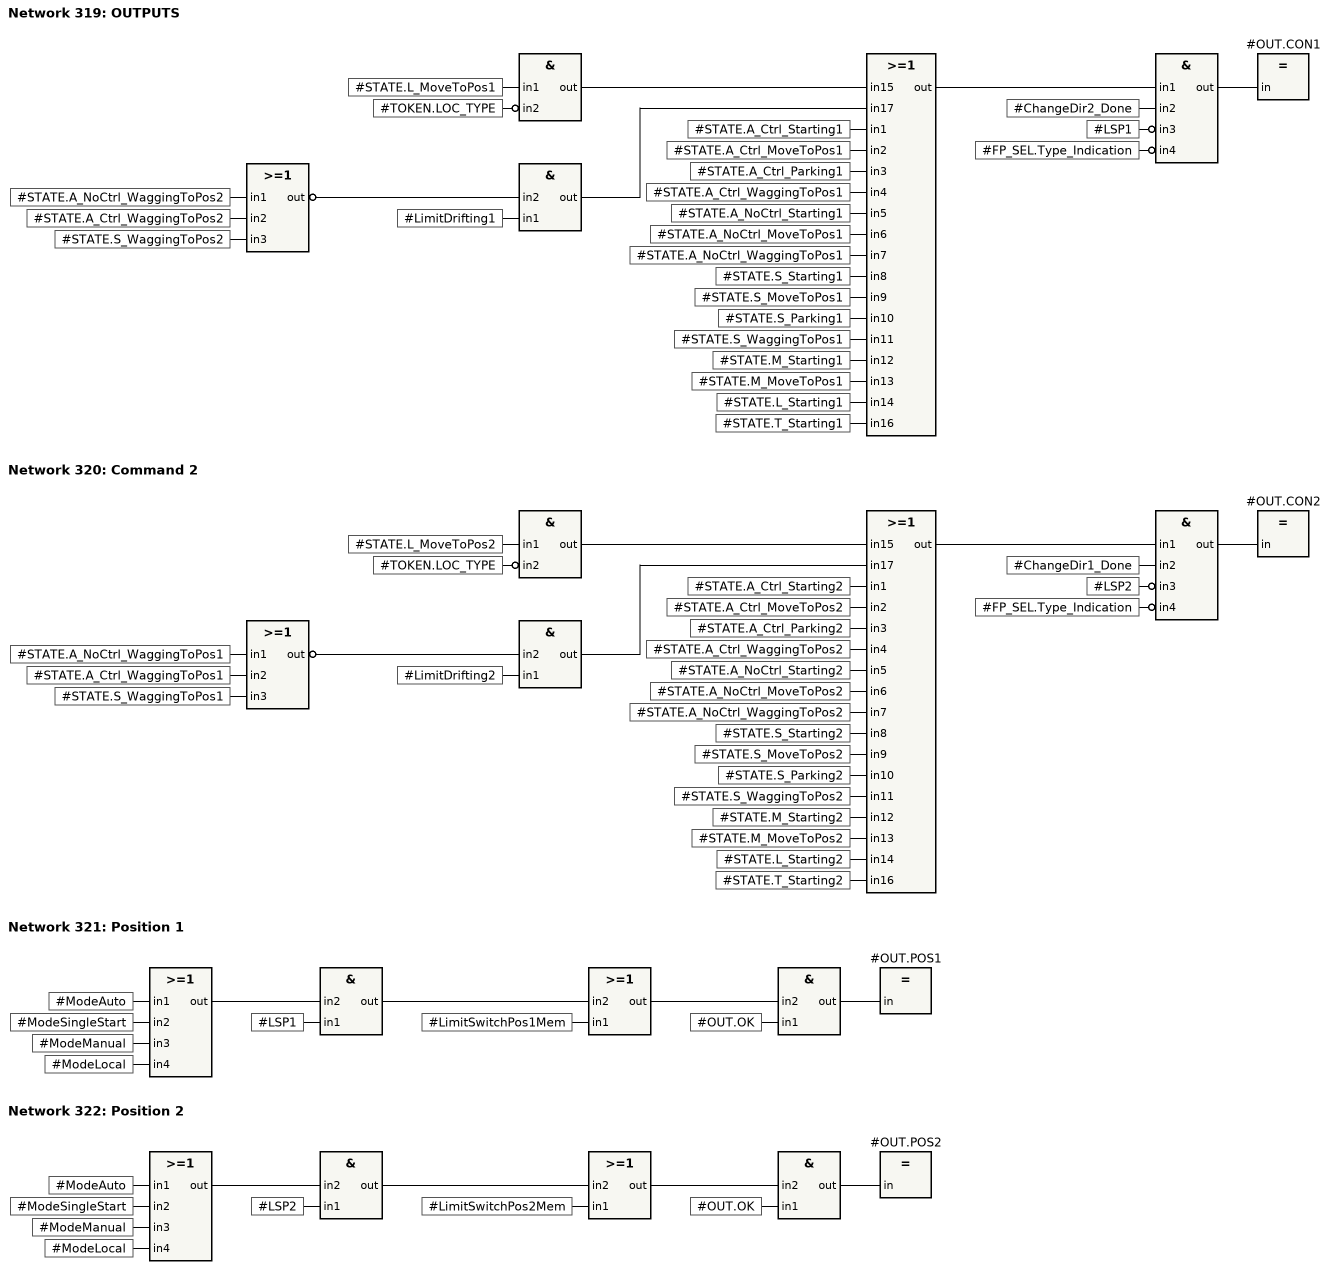
   #OUT.CON1 := ((#STATE.L_MoveToPos1 AND NOT #TOKEN.LOC_TYPE) OR (NOT (#STATE.A_NoCtrl_WaggingToPos2 OR #STATE.A_Ctrl_WaggingToPos2 OR #STATE.S_WaggingToPos2) AND #LimitDrifting1) OR #STATE.A_Ctrl_Starting1 OR #STATE.A_Ctrl_MoveToPos1 OR #STATE.A_Ctrl_Parking1 OR #STATE.A_Ctrl_WaggingToPos1 OR #STATE.A_NoCtrl_Starting1 OR #STATE.A_NoCtrl_MoveToPos1 OR #STATE.A_NoCtrl_WaggingToPos1 OR #STATE.S_Starting1 OR #STATE.S_MoveToPos1 OR #STATE.S_Parking1 OR #STATE.S_WaggingToPos1 OR #STATE.M_Starting1 OR #STATE.M_MoveToPos1 OR #STATE.L_Starting1 OR #STATE.T_Starting1) AND #ChangeDir2_Done AND NOT #LSP1 AND NOT #FP_SEL.Type_Indication;
END_REGION

REGION Network 320: Command 2
   // Build 003 - 2.July.2019 (EXTBOB): Added LOC_TYPE to prevent output being energized when running from the field
   #OUT.CON2 := ((#STATE.L_MoveToPos2 AND NOT #TOKEN.LOC_TYPE) OR (NOT (#STATE.A_NoCtrl_WaggingToPos1 OR #STATE.A_Ctrl_WaggingToPos1 OR #STATE.S_WaggingToPos1) AND #LimitDrifting2) OR #STATE.A_Ctrl_Starting2 OR #STATE.A_Ctrl_MoveToPos2 OR #STATE.A_Ctrl_Parking2 OR #STATE.A_Ctrl_WaggingToPos2 OR #STATE.A_NoCtrl_Starting2 OR #STATE.A_NoCtrl_MoveToPos2 OR #STATE.A_NoCtrl_WaggingToPos2 OR #STATE.S_Starting2 OR #STATE.S_MoveToPos2 OR #STATE.S_Parking2 OR #STATE.S_WaggingToPos2 OR #STATE.M_Starting2 OR #STATE.M_MoveToPos2 OR #STATE.L_Starting2 OR #STATE.T_Starting2) AND #ChangeDir1_Done AND NOT #LSP2 AND NOT #FP_SEL.Type_Indication;
END_REGION

REGION Network 321: Position 1
   #OUT.POS1 := (((#ModeAuto OR #ModeSingleStart OR #ModeManual OR #ModeLocal) AND #LSP1) OR #LimitSwitchPos1Mem) AND #OUT.OK;
END_REGION

REGION Network 322: Position 2
   #OUT.POS2 := (((#ModeAuto OR #ModeSingleStart OR #ModeManual OR #ModeLocal) AND #LSP2) OR #LimitSwitchPos2Mem) AND #OUT.OK;
END_REGION

REGION Network 323: OUTPUT
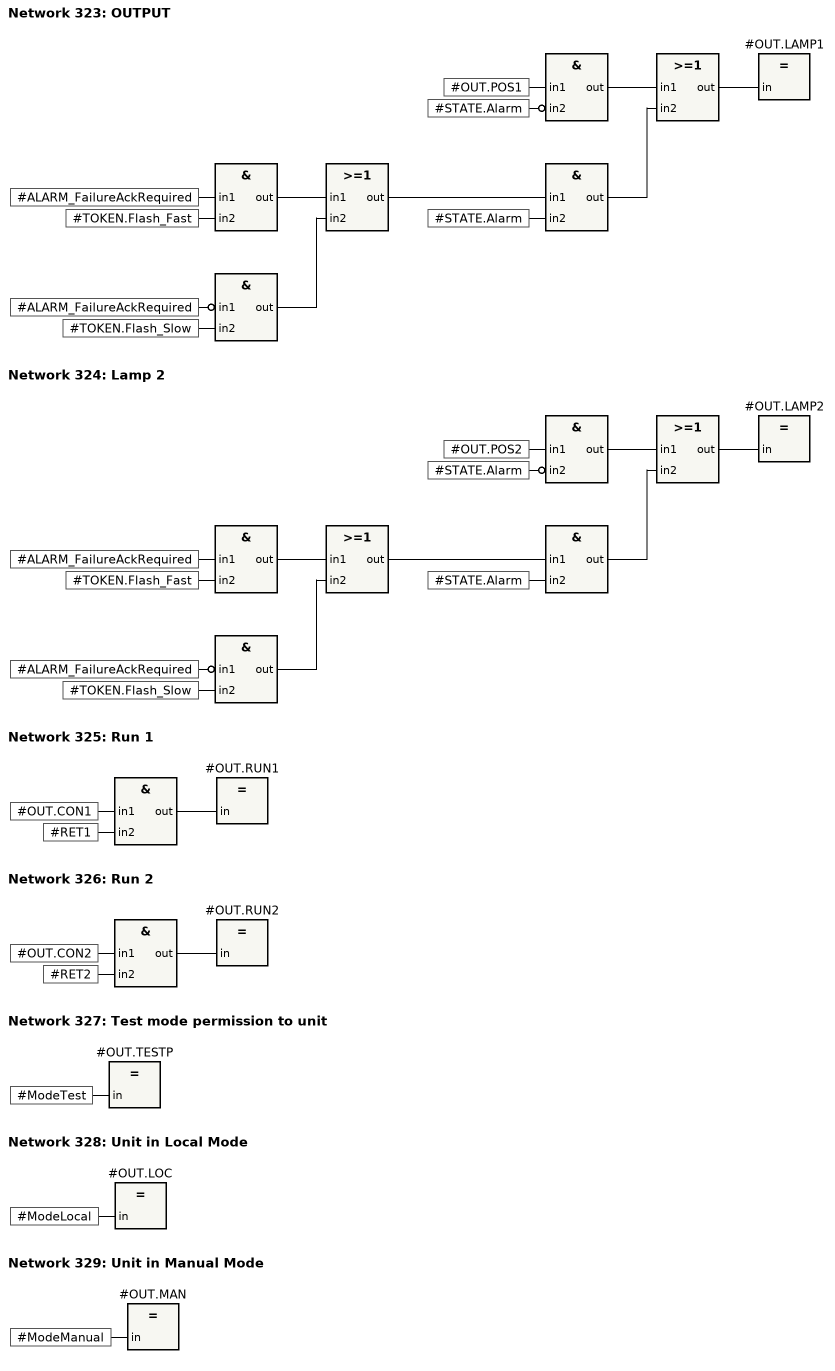
   #OUT.LAMP1 := (#OUT.POS1 AND NOT #STATE.Alarm) OR (((#ALARM_FailureAckRequired AND #TOKEN.Flash_Fast) OR (NOT #ALARM_FailureAckRequired AND #TOKEN.Flash_Slow)) AND #STATE.Alarm);
END_REGION

REGION Network 324: Lamp 2
   #OUT.LAMP2 := (#OUT.POS2 AND NOT #STATE.Alarm) OR (((#ALARM_FailureAckRequired AND #TOKEN.Flash_Fast) OR (NOT #ALARM_FailureAckRequired AND #TOKEN.Flash_Slow)) AND #STATE.Alarm);
END_REGION

REGION Network 325: Run 1
   #OUT.RUN1 := #OUT.CON1 AND #RET1;
END_REGION

REGION Network 326: Run 2
   #OUT.RUN2 := #OUT.CON2 AND #RET2;
END_REGION

REGION Network 327: Test mode permission to unit
   #OUT.TESTP := #ModeTest;
END_REGION

REGION Network 328: Unit in Local Mode
   #OUT.LOC := #ModeLocal;
END_REGION

REGION Network 329: Unit in Manual Mode
   #OUT.MAN := #ModeManual;
END_REGION

REGION Network 330: Unit in Auto Mode
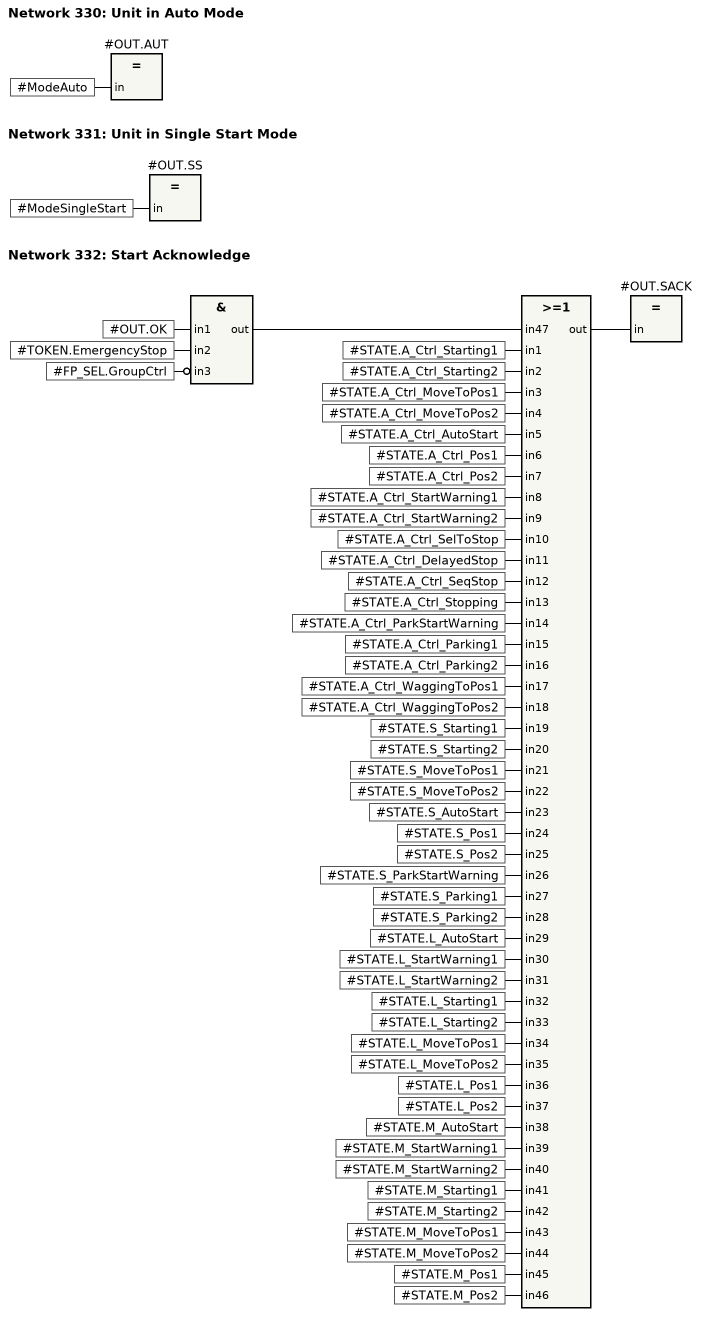
   #OUT.AUT := #ModeAuto;
END_REGION

REGION Network 331: Unit in Single Start Mode
   #OUT.SS := #ModeSingleStart;
END_REGION

REGION Network 332: Start Acknowledge
   #OUT.SACK := (#OUT.OK AND #TOKEN.EmergencyStop AND NOT #FP_SEL.GroupCtrl) OR #STATE.A_Ctrl_Starting1 OR #STATE.A_Ctrl_Starting2 OR #STATE.A_Ctrl_MoveToPos1 OR #STATE.A_Ctrl_MoveToPos2 OR #STATE.A_Ctrl_AutoStart OR #STATE.A_Ctrl_Pos1 OR #STATE.A_Ctrl_Pos2 OR #STATE.A_Ctrl_StartWarning1 OR #STATE.A_Ctrl_StartWarning2 OR #STATE.A_Ctrl_SelToStop OR #STATE.A_Ctrl_DelayedStop OR #STATE.A_Ctrl_SeqStop OR #STATE.A_Ctrl_Stopping OR #STATE.A_Ctrl_ParkStartWarning OR #STATE.A_Ctrl_Parking1 OR #STATE.A_Ctrl_Parking2 OR #STATE.A_Ctrl_WaggingToPos1 OR #STATE.A_Ctrl_WaggingToPos2 OR #STATE.S_Starting1 OR #STATE.S_Starting2 OR #STATE.S_MoveToPos1 OR #STATE.S_MoveToPos2 OR #STATE.S_AutoStart OR #STATE.S_Pos1 OR #STATE.S_Pos2 OR #STATE.S_ParkStartWarning OR #STATE.S_Parking1 OR #STATE.S_Parking2 OR #STATE.L_AutoStart OR #STATE.L_StartWarning1 OR #STATE.L_StartWarning2 OR #STATE.L_Starting1 OR #STATE.L_Starting2 OR #STATE.L_MoveToPos1 OR #STATE.L_MoveToPos2 OR #STATE.L_Pos1 OR #STATE.L_Pos2 OR #STATE.M_AutoStart OR #STATE.M_StartWarning1 OR #STATE.M_StartWarning2 OR #STATE.M_Starting1 OR #STATE.M_Starting2 OR #STATE.M_MoveToPos1 OR #STATE.M_MoveToPos2 OR #STATE.M_Pos1 OR #STATE.M_Pos2;
END_REGION

REGION Network 333
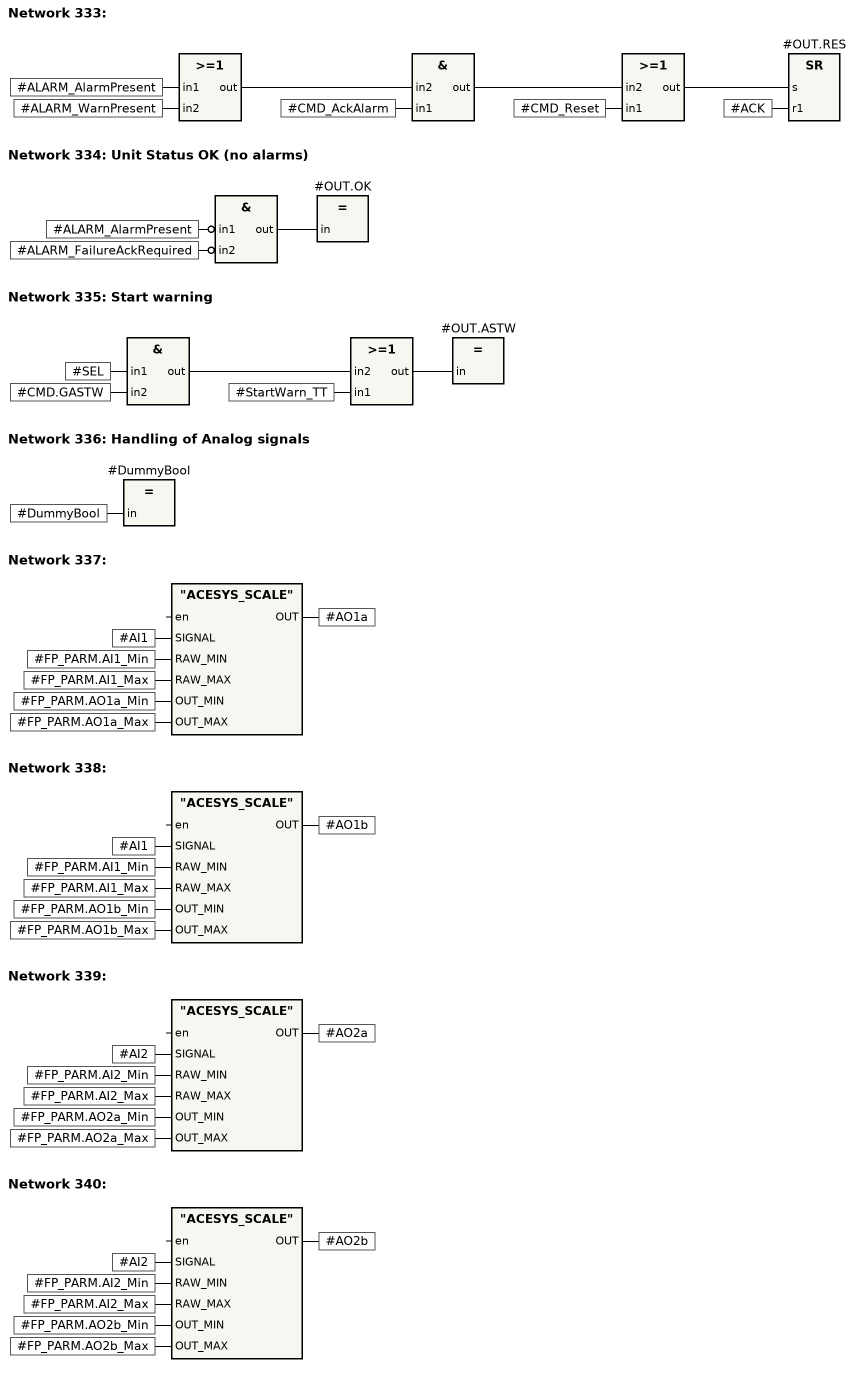
   IF ((#ALARM_AlarmPresent OR #ALARM_WarnPresent) AND #CMD_AckAlarm) OR #CMD_Reset THEN
       #OUT.RES := TRUE;   // SR flip-flop
   END_IF;
   IF #ACK THEN #OUT.RES := FALSE; END_IF;
END_REGION

REGION Network 334: Unit Status OK (no alarms)
   #OUT.OK := NOT #ALARM_AlarmPresent AND NOT #ALARM_FailureAckRequired;
END_REGION

REGION Network 335: Start warning
   #OUT.ASTW := (#SEL AND #CMD.GASTW) OR #StartWarn_TT;
END_REGION

REGION Network 336: Handling of Analog signals
   // ********************************************************************************
   // The block handles up to 3 analog signals.
   // 
   // The signals are AI1, AI2 and AI3 they are defined as reals.
   // 
   // By configuration at runtime these analog signals are converted into each 2 
   // values.
   // 
   // The parametres given from ECS defines:
   // 
   // 1) Min and Max for the input signal
   // 2) Corresponding Min and Max for Analog output "a"
   // 3) Corresponding Min and Max for Analog output "b"
   // 
   // Output a and b can be used for for instance a value in % and one in engineering 
   // units.
   // 
   // An example could be:
   // A motor current with a norminal value of 75 A
   // Input : motor current in mA; min=0, max = 75000
   // 
   // The signals are calculated by defining the formula for the line
   // 
   // Y = aX+b
   // 
   // Where a = (Y2 - Y1)/(X2-X1)
   // and   b = Y2 - aX2
   // Output a : motor current in %; min = 0, max = 100
   // output b : motor current in A; min = 0, max = 75
   #DummyBool := #DummyBool;
END_REGION

REGION Network 337
   "ACESYS_SCALE"(SIGNAL := #AI1,
                  RAW_MIN := #FP_PARM.AI1_Min,
                  RAW_MAX := #FP_PARM.AI1_Max,
                  OUT_MIN := #FP_PARM.AO1a_Min,
                  OUT_MAX := #FP_PARM.AO1a_Max,
                  OUT => #AO1a);
END_REGION

REGION Network 338
   "ACESYS_SCALE"(SIGNAL := #AI1,
                  RAW_MIN := #FP_PARM.AI1_Min,
                  RAW_MAX := #FP_PARM.AI1_Max,
                  OUT_MIN := #FP_PARM.AO1b_Min,
                  OUT_MAX := #FP_PARM.AO1b_Max,
                  OUT => #AO1b);
END_REGION

REGION Network 339
   "ACESYS_SCALE"(SIGNAL := #AI2,
                  RAW_MIN := #FP_PARM.AI2_Min,
                  RAW_MAX := #FP_PARM.AI2_Max,
                  OUT_MIN := #FP_PARM.AO2a_Min,
                  OUT_MAX := #FP_PARM.AO2a_Max,
                  OUT => #AO2a);
END_REGION

REGION Network 340
   "ACESYS_SCALE"(SIGNAL := #AI2,
                  RAW_MIN := #FP_PARM.AI2_Min,
                  RAW_MAX := #FP_PARM.AI2_Max,
                  OUT_MIN := #FP_PARM.AO2b_Min,
                  OUT_MAX := #FP_PARM.AO2b_Max,
                  OUT => #AO2b);
END_REGION

REGION Network 341
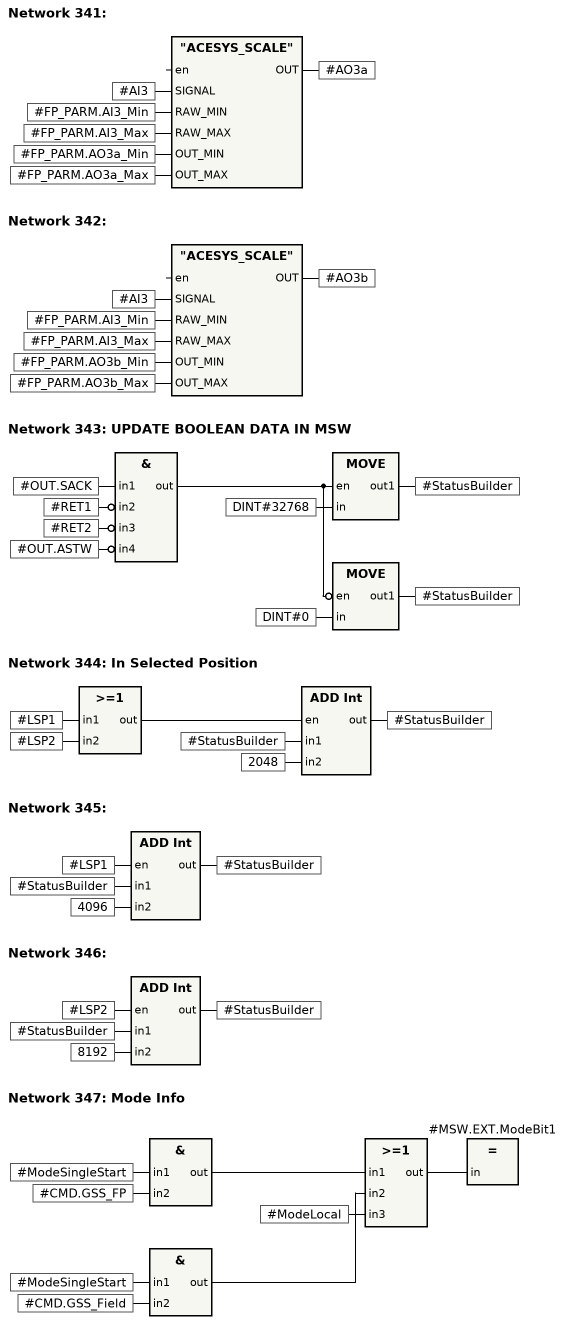
   "ACESYS_SCALE"(SIGNAL := #AI3,
                  RAW_MIN := #FP_PARM.AI3_Min,
                  RAW_MAX := #FP_PARM.AI3_Max,
                  OUT_MIN := #FP_PARM.AO3a_Min,
                  OUT_MAX := #FP_PARM.AO3a_Max,
                  OUT => #AO3a);
END_REGION

REGION Network 342
   "ACESYS_SCALE"(SIGNAL := #AI3,
                  RAW_MIN := #FP_PARM.AI3_Min,
                  RAW_MAX := #FP_PARM.AI3_Max,
                  OUT_MIN := #FP_PARM.AO3b_Min,
                  OUT_MAX := #FP_PARM.AO3b_Max,
                  OUT => #AO3b);
END_REGION

REGION Network 343: UPDATE BOOLEAN DATA IN MSW
   #_w1 := #OUT.SACK AND NOT #RET1 AND NOT #RET2 AND NOT #OUT.ASTW;
   IF #_w1 THEN #StatusBuilder := DINT#32768; END_IF;
   IF NOT #_w1 THEN #StatusBuilder := DINT#0; END_IF;
END_REGION

REGION Network 344: In Selected Position
   // Build 002: 26 March 2019 : Direction request removed to show selected position
   IF #LSP1 OR #LSP2 THEN #StatusBuilder := #StatusBuilder + 2048; END_IF;
END_REGION

REGION Network 345
   IF #LSP1 THEN #StatusBuilder := #StatusBuilder + 4096; END_IF;
END_REGION

REGION Network 346
   IF #LSP2 THEN #StatusBuilder := #StatusBuilder + 8192; END_IF;
END_REGION

REGION Network 347: Mode Info
   #MSW.EXT.ModeBit1 := (#ModeSingleStart AND #CMD.GSS_FP) OR (#ModeSingleStart AND #CMD.GSS_Field) OR #ModeLocal;
END_REGION

REGION Network 348: Mode Info
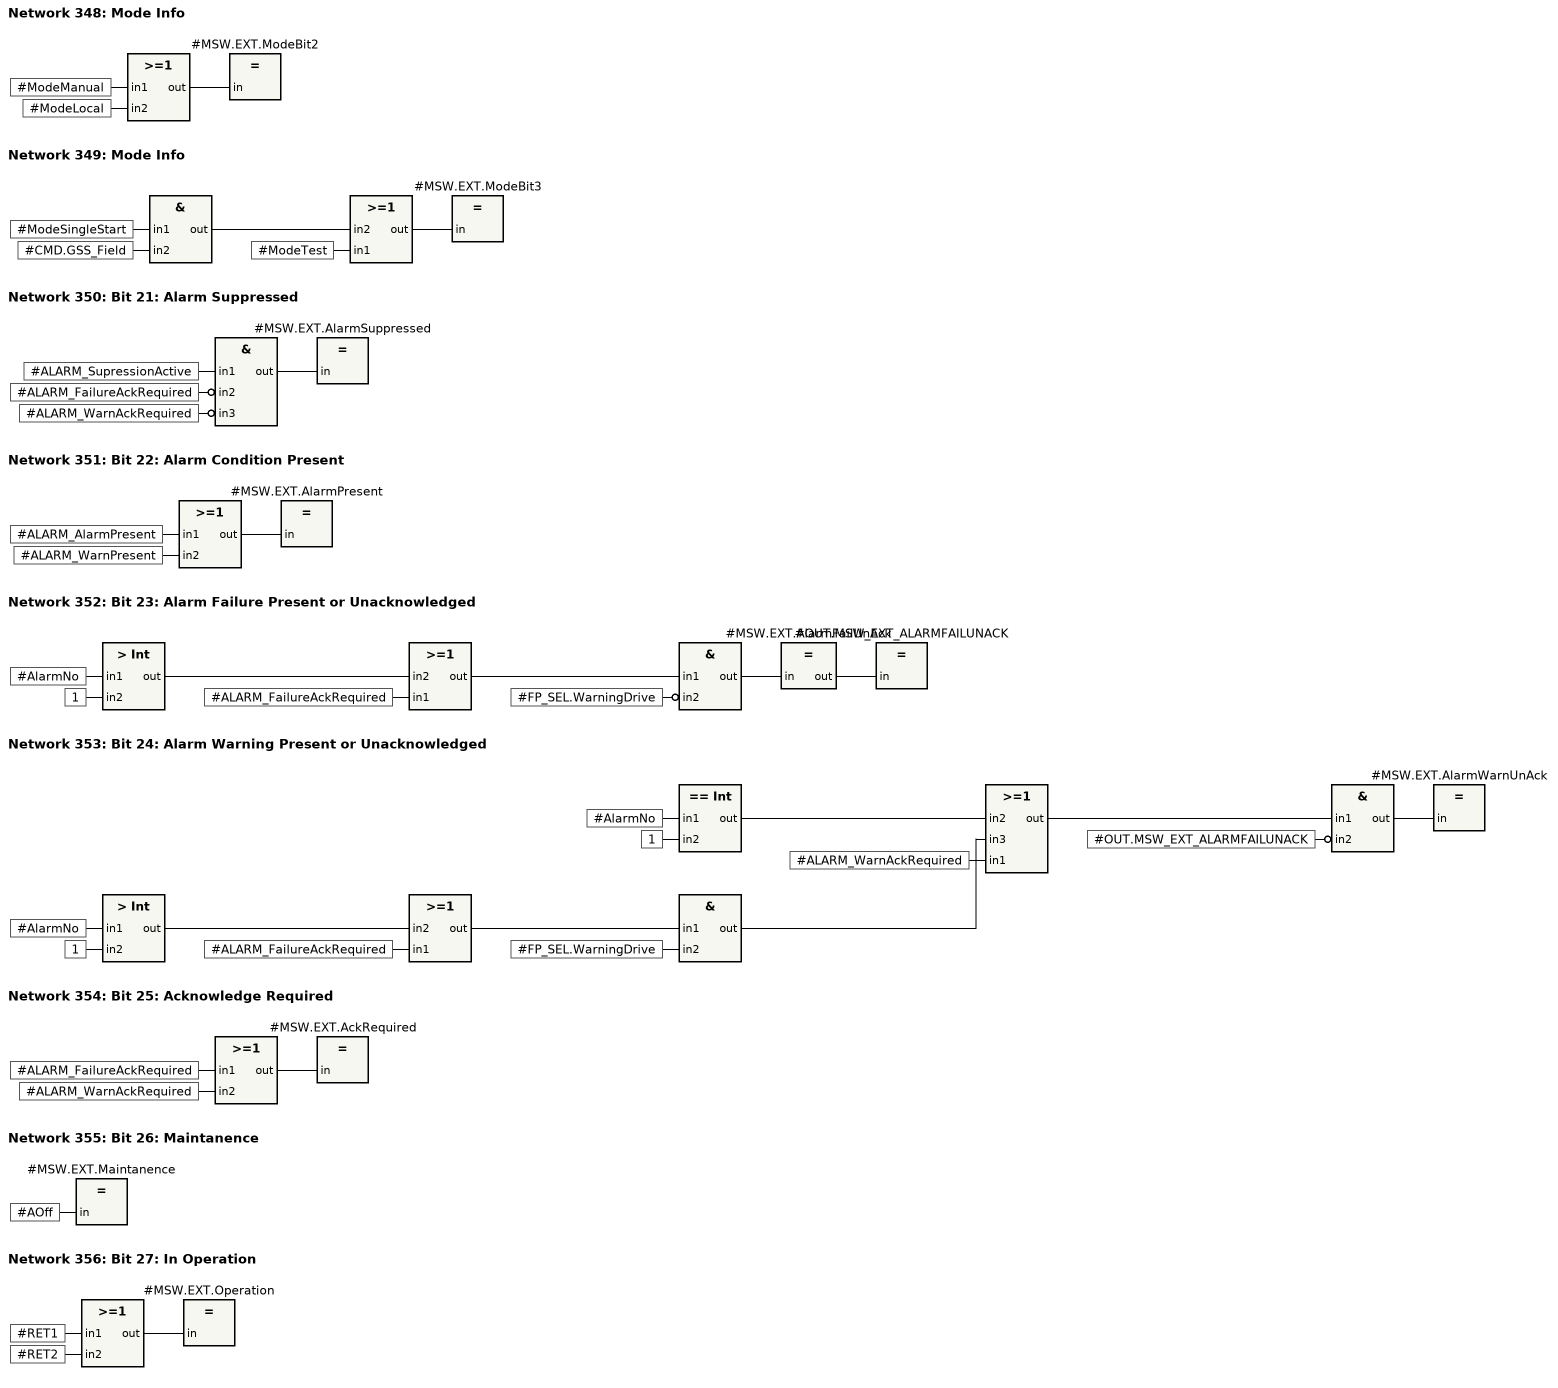
   #MSW.EXT.ModeBit2 := #ModeManual OR #ModeLocal;
END_REGION

REGION Network 349: Mode Info
   #MSW.EXT.ModeBit3 := (#ModeSingleStart AND #CMD.GSS_Field) OR #ModeTest;
END_REGION

REGION Network 350: Bit 21: Alarm Suppressed
   #MSW.EXT.AlarmSuppressed := #ALARM_SupressionActive AND NOT #ALARM_FailureAckRequired AND NOT #ALARM_WarnAckRequired;
END_REGION

REGION Network 351: Bit 22: Alarm Condition Present
   #MSW.EXT.AlarmPresent := #ALARM_AlarmPresent OR #ALARM_WarnPresent;
END_REGION

REGION Network 352: Bit 23: Alarm Failure Present or Unacknowledged
   #MSW.EXT.AlarmFailUnAck := ((#AlarmNo > 1) OR #ALARM_FailureAckRequired) AND NOT #FP_SEL.WarningDrive;
   #OUT.MSW_EXT_ALARMFAILUNACK := #MSW.EXT.AlarmFailUnAck;
END_REGION

REGION Network 353: Bit 24: Alarm Warning Present or Unacknowledged
   #MSW.EXT.AlarmWarnUnAck := ((#AlarmNo = 1) OR (((#AlarmNo > 1) OR #ALARM_FailureAckRequired) AND #FP_SEL.WarningDrive) OR #ALARM_WarnAckRequired) AND NOT #OUT.MSW_EXT_ALARMFAILUNACK;
END_REGION

REGION Network 354: Bit 25: Acknowledge Required
   #MSW.EXT.AckRequired := #ALARM_FailureAckRequired OR #ALARM_WarnAckRequired;
END_REGION

REGION Network 355: Bit 26: Maintanence
   #MSW.EXT.Maintanence := #AOff;
END_REGION

REGION Network 356: Bit 27: In Operation
   #MSW.EXT.Operation := #RET1 OR #RET2;
END_REGION

REGION Network 357: Bit 28: Forced
   // Build 002: 26 March 2019 : OutOfService flag will set bit 28 to enable force icon
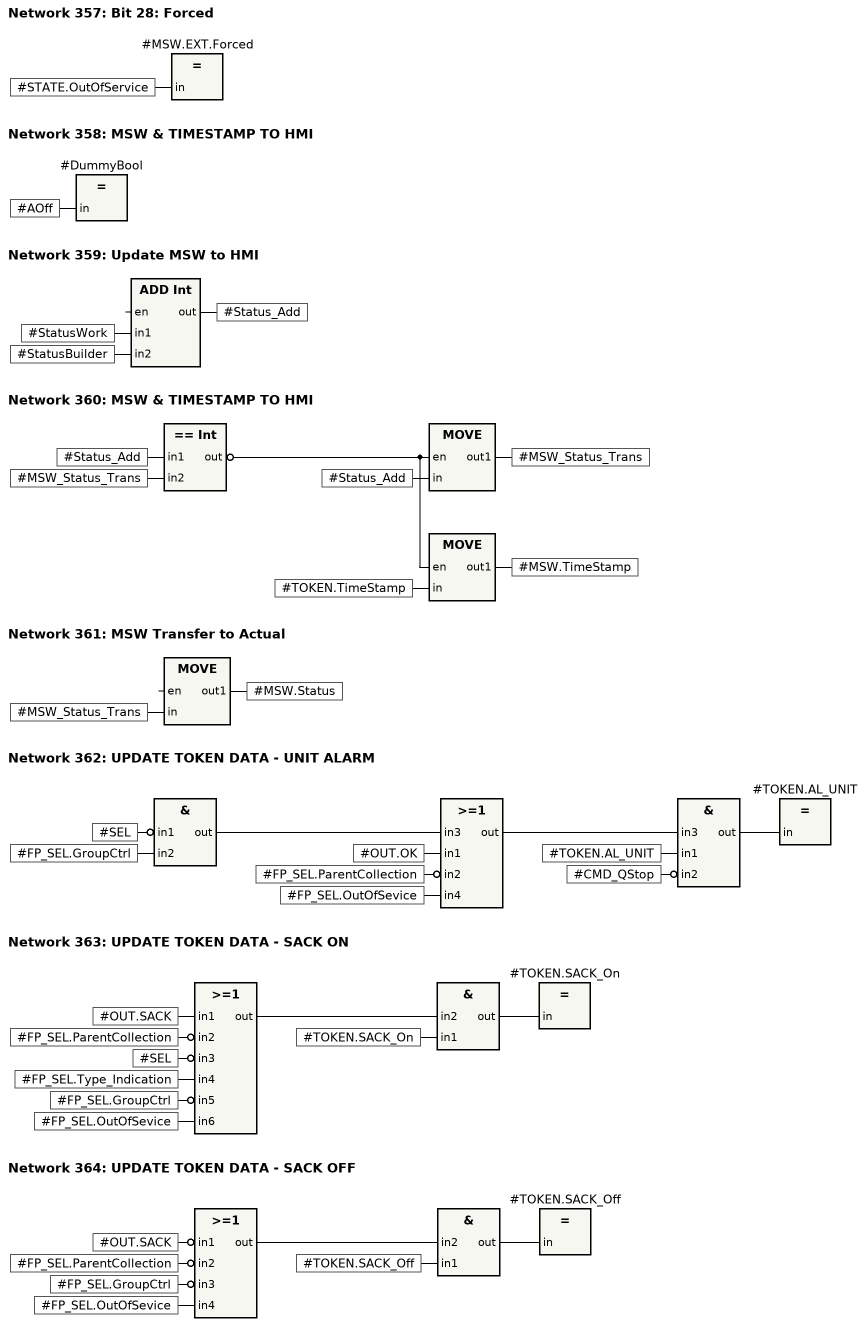
   #MSW.EXT.Forced := #STATE.OutOfService;
END_REGION

REGION Network 358: MSW & TIMESTAMP TO HMI
   Done:
   #DummyBool := #AOff;
END_REGION

REGION Network 359: Update MSW to HMI
   #Status_Add := #StatusWork + #StatusBuilder;
END_REGION

REGION Network 360: MSW & TIMESTAMP TO HMI
   #_w1 := NOT (#Status_Add = #MSW_Status_Trans);
   IF #_w1 THEN
       #MSW_Status_Trans := #Status_Add;
       #MSW.TimeStamp := #TOKEN.TimeStamp;
   END_IF;
END_REGION

REGION Network 361: MSW Transfer to Actual
   #MSW.Status := #MSW_Status_Trans;
END_REGION

REGION Network 362: UPDATE TOKEN DATA - UNIT ALARM
   #TOKEN.AL_UNIT := ((NOT #SEL AND #FP_SEL.GroupCtrl) OR #OUT.OK OR NOT #FP_SEL.ParentCollection OR #FP_SEL.OutOfSevice) AND #TOKEN.AL_UNIT AND NOT #CMD_QStop;
END_REGION

REGION Network 363: UPDATE TOKEN DATA - SACK ON
   // Build 003 - 02.July.2019 (EXTBOB): Replaced "Select" with original explicit definition
   // Build 007 - 24.Jun.2020 (MIA-US): Removed CMD.GSEL
   #TOKEN.SACK_On := (#OUT.SACK OR NOT #FP_SEL.ParentCollection OR NOT #SEL OR #FP_SEL.Type_Indication OR NOT #FP_SEL.GroupCtrl OR #FP_SEL.OutOfSevice) AND #TOKEN.SACK_On;
END_REGION

REGION Network 364: UPDATE TOKEN DATA - SACK OFF
   #TOKEN.SACK_Off := (NOT #OUT.SACK OR NOT #FP_SEL.ParentCollection OR NOT #FP_SEL.GroupCtrl OR #FP_SEL.OutOfSevice) AND #TOKEN.SACK_Off;
END_REGION

REGION Network 365: UPDATE TOKEN DATA - ALL UNITS AUTO
   // Build 003 - 02.July.2019 (EXTBOB): Replaced "Select" with original explicit definition
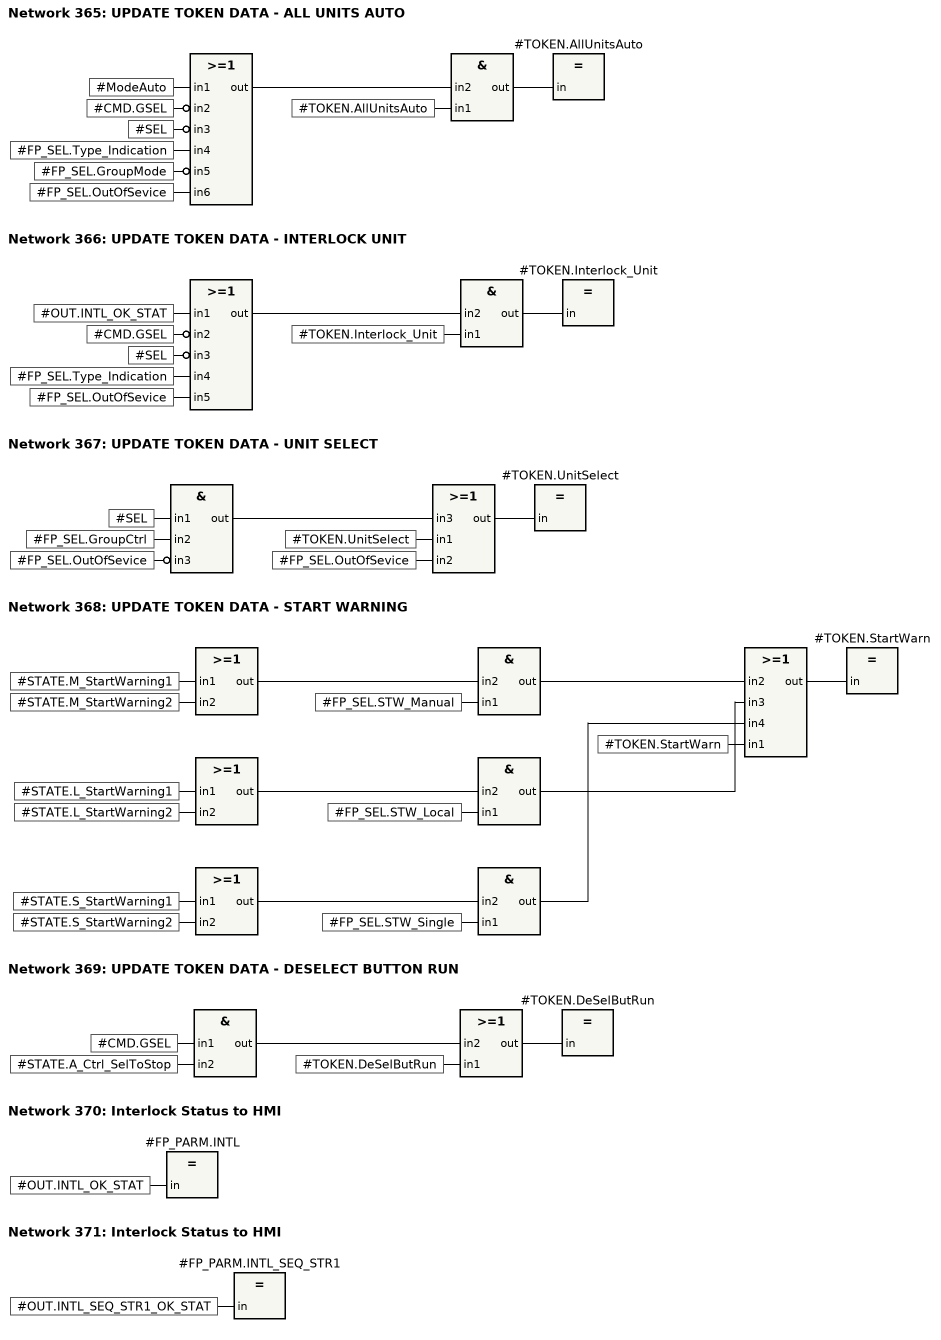
   #TOKEN.AllUnitsAuto := (#ModeAuto OR NOT #CMD.GSEL OR NOT #SEL OR #FP_SEL.Type_Indication OR NOT #FP_SEL.GroupMode OR #FP_SEL.OutOfSevice) AND #TOKEN.AllUnitsAuto;
END_REGION

REGION Network 366: UPDATE TOKEN DATA - INTERLOCK UNIT
   // Build 003 - 02.July.2019 (EXTBOB): Replaced "Select" with original explicit definition
   #TOKEN.Interlock_Unit := (#OUT.INTL_OK_STAT OR NOT #CMD.GSEL OR NOT #SEL OR #FP_SEL.Type_Indication OR #FP_SEL.OutOfSevice) AND #TOKEN.Interlock_Unit;
END_REGION

REGION Network 367: UPDATE TOKEN DATA - UNIT SELECT
   #TOKEN.UnitSelect := (#SEL AND #FP_SEL.GroupCtrl AND NOT #FP_SEL.OutOfSevice) OR #TOKEN.UnitSelect OR #FP_SEL.OutOfSevice;
END_REGION

REGION Network 368: UPDATE TOKEN DATA - START WARNING
   #TOKEN.StartWarn := ((#STATE.M_StartWarning1 OR #STATE.M_StartWarning2) AND #FP_SEL.STW_Manual) OR ((#STATE.L_StartWarning1 OR #STATE.L_StartWarning2) AND #FP_SEL.STW_Local) OR ((#STATE.S_StartWarning1 OR #STATE.S_StartWarning2) AND #FP_SEL.STW_Single) OR #TOKEN.StartWarn;
END_REGION

REGION Network 369: UPDATE TOKEN DATA - DESELECT BUTTON RUN
   #TOKEN.DeSelButRun := (#CMD.GSEL AND #STATE.A_Ctrl_SelToStop) OR #TOKEN.DeSelButRun;
END_REGION

REGION Network 370: Interlock Status to HMI
   #FP_PARM.INTL := #OUT.INTL_OK_STAT;
END_REGION

REGION Network 371: Interlock Status to HMI
   #FP_PARM.INTL_SEQ_STR1 := #OUT.INTL_SEQ_STR1_OK_STAT;
END_REGION

REGION Network 372: Interlock Status to HMI
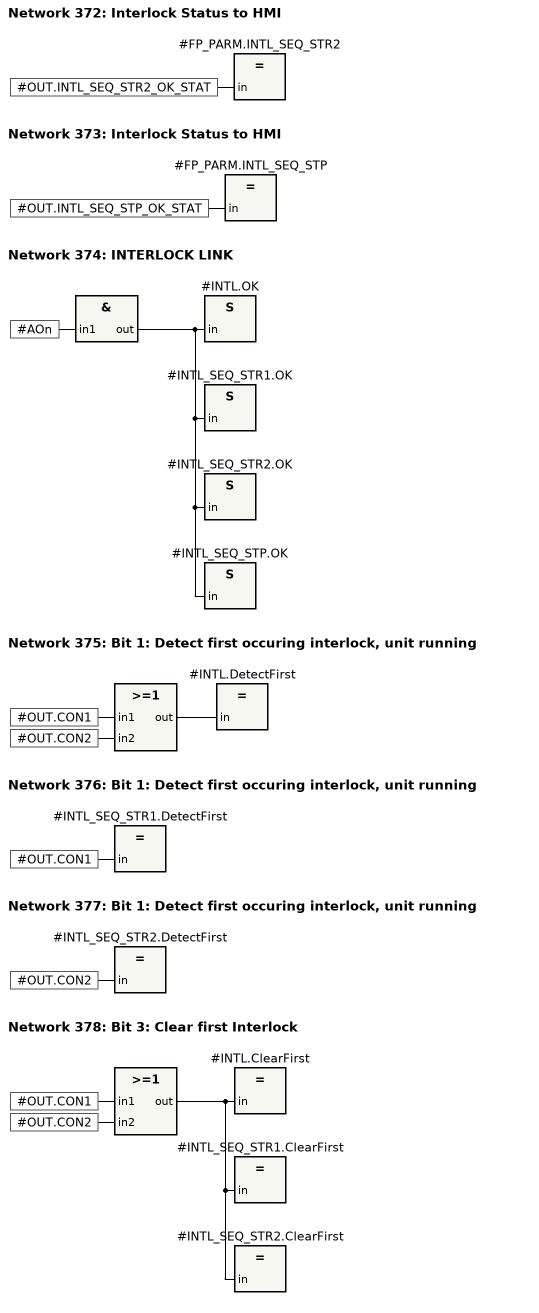
   #FP_PARM.INTL_SEQ_STR2 := #OUT.INTL_SEQ_STR2_OK_STAT;
END_REGION

REGION Network 373: Interlock Status to HMI
   #FP_PARM.INTL_SEQ_STP := #OUT.INTL_SEQ_STP_OK_STAT;
END_REGION

REGION Network 374: INTERLOCK LINK
   IF #AOn THEN
       #INTL.OK := TRUE;
       #INTL_SEQ_STR1.OK := TRUE;
       #INTL_SEQ_STR2.OK := TRUE;
       #INTL_SEQ_STP.OK := TRUE;
   END_IF;
END_REGION

REGION Network 375: Bit 1: Detect first occuring interlock, unit running
   #INTL.DetectFirst := #OUT.CON1 OR #OUT.CON2;
END_REGION

REGION Network 376: Bit 1: Detect first occuring interlock, unit running
   #INTL_SEQ_STR1.DetectFirst := #OUT.CON1;
END_REGION

REGION Network 377: Bit 1: Detect first occuring interlock, unit running
   #INTL_SEQ_STR2.DetectFirst := #OUT.CON2;
END_REGION

REGION Network 378: Bit 3: Clear first Interlock
   #INTL.ClearFirst := #OUT.CON1 OR #OUT.CON2;
   #INTL_SEQ_STR1.ClearFirst := #INTL.ClearFirst;
   #INTL_SEQ_STR2.ClearFirst := #INTL.ClearFirst;
END_REGION

REGION Network 379: DEVICE SIMULATION
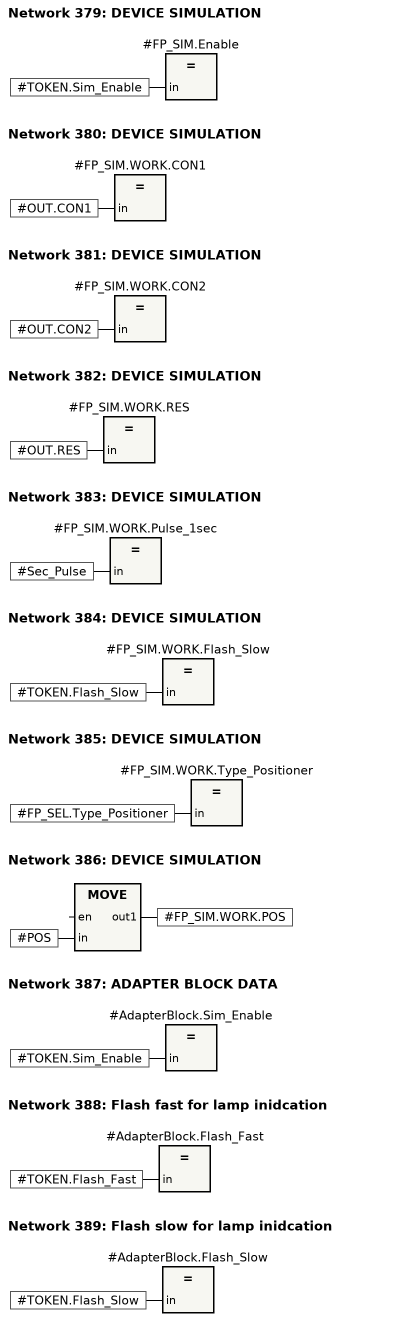
   #FP_SIM.Enable := #TOKEN.Sim_Enable;
END_REGION

REGION Network 380: DEVICE SIMULATION
   #FP_SIM.WORK.CON1 := #OUT.CON1;
END_REGION

REGION Network 381: DEVICE SIMULATION
   #FP_SIM.WORK.CON2 := #OUT.CON2;
END_REGION

REGION Network 382: DEVICE SIMULATION
   #FP_SIM.WORK.RES := #OUT.RES;
END_REGION

REGION Network 383: DEVICE SIMULATION
   #FP_SIM.WORK.Pulse_1sec := #Sec_Pulse;
END_REGION

REGION Network 384: DEVICE SIMULATION
   #FP_SIM.WORK.Flash_Slow := #TOKEN.Flash_Slow;
END_REGION

REGION Network 385: DEVICE SIMULATION
   #FP_SIM.WORK.Type_Positioner := #FP_SEL.Type_Positioner;
END_REGION

REGION Network 386: DEVICE SIMULATION
   #FP_SIM.WORK.POS := #POS;
END_REGION

REGION Network 387: ADAPTER BLOCK DATA
   #AdapterBlock.Sim_Enable := #TOKEN.Sim_Enable;
END_REGION

REGION Network 388: Flash fast for lamp inidcation
   #AdapterBlock.Flash_Fast := #TOKEN.Flash_Fast;
END_REGION

REGION Network 389: Flash slow for lamp inidcation
   #AdapterBlock.Flash_Slow := #TOKEN.Flash_Slow;
END_REGION

REGION Network 390: 1 Seconds Puls
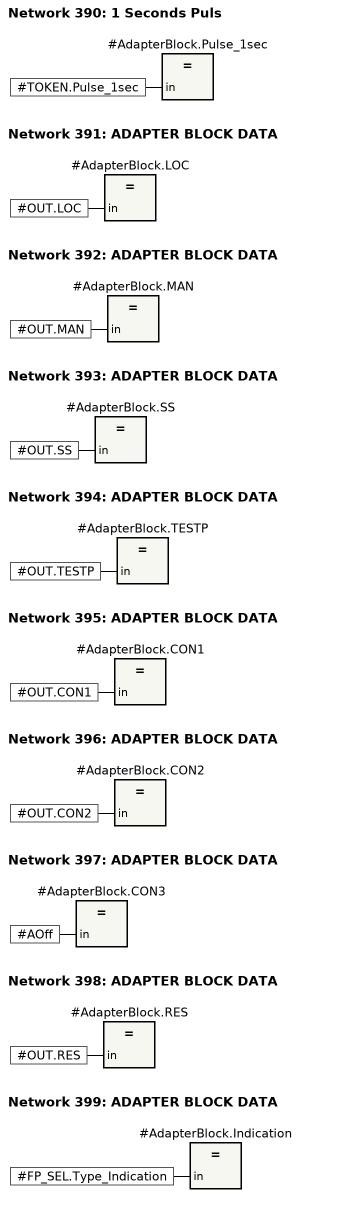
   #AdapterBlock.Pulse_1sec := #TOKEN.Pulse_1sec;
END_REGION

REGION Network 391: ADAPTER BLOCK DATA
   #AdapterBlock.LOC := #OUT.LOC;
END_REGION

REGION Network 392: ADAPTER BLOCK DATA
   #AdapterBlock.MAN := #OUT.MAN;
END_REGION

REGION Network 393: ADAPTER BLOCK DATA
   #AdapterBlock.SS := #OUT.SS;
END_REGION

REGION Network 394: ADAPTER BLOCK DATA
   #AdapterBlock.TESTP := #OUT.TESTP;
END_REGION

REGION Network 395: ADAPTER BLOCK DATA
   #AdapterBlock.CON1 := #OUT.CON1;
END_REGION

REGION Network 396: ADAPTER BLOCK DATA
   #AdapterBlock.CON2 := #OUT.CON2;
END_REGION

REGION Network 397: ADAPTER BLOCK DATA
   #AdapterBlock.CON3 := #AOff;
END_REGION

REGION Network 398: ADAPTER BLOCK DATA
   #AdapterBlock.RES := #OUT.RES;
END_REGION

REGION Network 399: ADAPTER BLOCK DATA
   #AdapterBlock.Indication := #FP_SEL.Type_Indication;
END_REGION

REGION Network 400: Write STAT to OUT
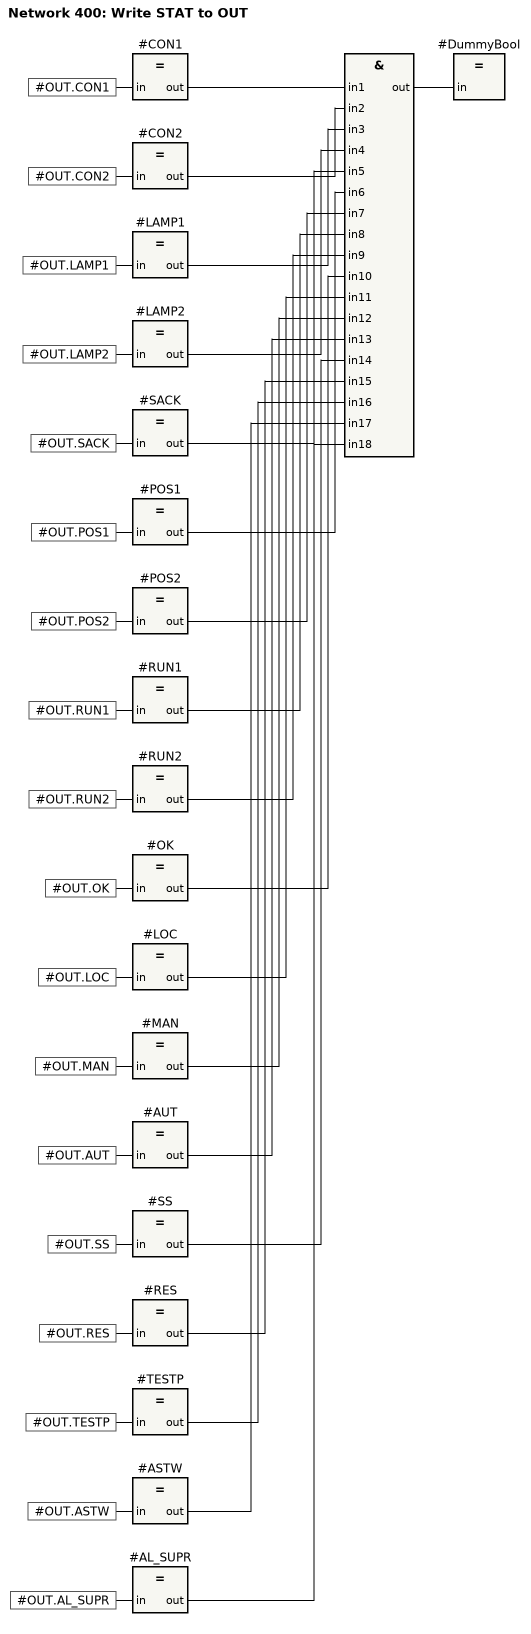
   #CON1 := #OUT.CON1;
   #CON2 := #OUT.CON2;
   #LAMP1 := #OUT.LAMP1;
   #LAMP2 := #OUT.LAMP2;
   #SACK := #OUT.SACK;
   #POS1 := #OUT.POS1;
   #POS2 := #OUT.POS2;
   #RUN1 := #OUT.RUN1;
   #RUN2 := #OUT.RUN2;
   #OK := #OUT.OK;
   #LOC := #OUT.LOC;
   #MAN := #OUT.MAN;
   #AUT := #OUT.AUT;
   #SS := #OUT.SS;
   #RES := #OUT.RES;
   #TESTP := #OUT.TESTP;
   #ASTW := #OUT.ASTW;
   #AL_SUPR := #OUT.AL_SUPR;
   #DummyBool := #OUT.CON1 AND #OUT.CON2 AND #OUT.LAMP1 AND #OUT.LAMP2 AND #OUT.SACK AND #OUT.POS1 AND #OUT.POS2 AND #OUT.RUN1 AND #OUT.RUN2 AND #OUT.OK AND #OUT.LOC AND #OUT.MAN AND #OUT.AUT AND #OUT.SS AND #OUT.RES AND #OUT.TESTP AND #OUT.ASTW AND #OUT.AL_SUPR;
END_REGION
END_FUNCTION_BLOCK

FUNCTION_BLOCK "ACESYS_VALVE"   // FB212, FBD
TITLE = ACESYS V8.0 - Build 001 - VALVE Block / ACESYS V8.0 - Build 008 - VALVE Block
{ S7_Optimized_Access := 'FALSE' }
AUTHOR : FLSmidth
FAMILY : ACESYS
NAME : VALVE
VERSION : 8.0
   VAR_INPUT
      CMD : "ACESYS_GRP_CMD";
      SEL : Bool := TRUE;   // Unit Select by User program
      PREQ1 : Bool := TRUE;   // Direction 1 Select
      PREQ2 : Bool := TRUE;   // Direction 2 Select
      PREQ3 : Bool := TRUE;   // Direction 3 Select
      RDY : Bool := TRUE;   // Unit ready
      OVL : Bool := TRUE;   // Overload / trip
      LSP1 : Bool;   // Limit Switch Pos 1
      LSP2 : Bool;   // Limit Switch Pos 2
      LSP3 : Bool;   // Limit Switch Pos 3
      LSTR1 : Bool;   // Local start 1
      LSTR2 : Bool;   // Local start 2
      LSTR3 : Bool;   // Local start 3
      REM : Bool := TRUE;   // Unit in Remote operation
      SSW : Bool := TRUE;   // Safety switch
      DRDY : Bool := TRUE;   // Drive / MCC ready
      GFA : Bool := TRUE;   // General fault
      GWA : Bool := TRUE;   // General waring
      BUSF : Bool := TRUE;   // Bus failure
      UTEST : Bool;   // Drawer in test position
      ACK : Bool;   // Feedback from unit on alarm reset
      AI1 : Real;   // Analog value 1
      AI2 : Real;   // Analog value 2
      AI3 : Real;   // Abalog value 3
   END_VAR
   VAR_OUTPUT
      INTL : "ACESYS_INTL";   // Interlock
      INTL_SEQ_STR1 : "ACESYS_INTL";   // Interlock Sequence Start Dir 1
      INTL_SEQ_STR2 : "ACESYS_INTL";   // Interlock Sequence Start Dir 2
      INTL_SEQ_STR3 : "ACESYS_INTL";   // Interlock Sequence Start Dir 3
      INTL_SEQ_STP : "ACESYS_INTL";   // Interlock Sequence Stop
      CON1 : Bool;   // Command 1
      CON2 : Bool;   // Command 2
      CON3 : Bool;   // Command 3
      LAMP1 : Bool;   // Lamp 1
      LAMP2 : Bool;   // Lamp 2
      LAMP3 : Bool;   // Lamp 3
      SACK : Bool;   // Start Acknowledge
      POS1 : Bool;   // Position 1
      POS2 : Bool;   // Position 2
      POS3 : Bool;   // Position 2
      OK : Bool;   // Unit Status OK (no alarms)
      LOC : Bool;   // Unit in Local Mode
      MAN : Bool;   // Unit in Manual Mode
      AUT : Bool;   // Unit in Auto Mode
      SS : Bool;   // Unit in Single Start Mode
      RES : Bool;   // Reset to unit
      TESTP : Bool;   // Test mode permission to unit
      ASTW : Bool;   // Start warning
      AL_SUPR : Bool;   // Supress Child Alarms
      AO1a : Real;   // Analog converted 1a
      AO1b : Real;   // Analog converted 1b
      AO2a : Real;   // Analog converted 2a
      AO2b : Real;   // Analog converted 2b
      AO3a : Real;   // Analog converted 3a
      AO3b : Real;   // Analog converted 3b
      MSW : "ACESYS_HMI_STAT_32T";
   END_VAR
   VAR_IN_OUT
      TOKEN : "ACESYS_TOKEN";
   END_VAR
   VAR
      BlockInfo : Struct
         Ace_Version : Int;   // Acesys Block Version Number
         Ace_BuildNo : Int;   // Acesys Block Build Number
         State_Act : Int;   // Actual State Number
         State_Prev : Int;   // Previous State Number
         DB_Number : Int;   // Block Instance DB Number
      END_STRUCT;
      FP_CMD : Struct   // Faceplate Commands
         Test : Bool;
         QuickStop : Bool;
         Spare_09 : Bool;
         Spare_10 : Bool;
         Spare_11 : Bool;
         Spare_12 : Bool;
         Spare_13 : Bool;
         AckAlarm : Bool;
         Auto : Bool;
         Manual : Bool;
         Local : Bool;
         Start1 : Bool;
         Start2 : Bool;
         Start3 : Bool;
         Stop : Bool;
         Reset : Bool;
      END_STRUCT;
      FP_SEL : Struct   // Faceplate Selections
         STW_AutoStart : Bool;   // Faceplate Start Warning in Auto Start mode
         STW_Local : Bool;   // Faceplate Start Warning in Local mode
         STW_Manual : Bool;   // Faceplate Start Warning in Manual mode
         STW_Single : Bool;   // Faceplate Start Warning in Single Start mode
         Type_2Pos : Bool;   // Faceplate Motorgate type
         Type_3Pos : Bool;   // Faceplate Positioner type
         Type_Indication : Bool;   // Faceplate Indication type
         Type_NoLimit : Bool;   // Faceplate Indication type
         Type_ConstantCmd : Bool;   // Faceplate Indication type
         Type_PulseCmd : Bool;   // Faceplate Indication type
         ParentSupress : Bool;   // Enable Parent Supress of alarms
         ParentCollection : Bool;   // Enable Inching in Manual Mode
         INCH_Man : Bool;   // Enable Inching in Manual Mode
         INCH_Loc : Bool;   // Enable Inching in Local Mode
         OutOfSevice : Bool;   // Select Out of Service
         WarningDrive : Bool;   // 0 = Failure Drive / 1 = Warning Drive
         Park_CurrPos : Bool;
         Park_Pos1 : Bool;
         Park_Pos2 : Bool;
         Park_Pos3 : Bool;
         GroupMode : Bool;
         GroupCtrl : Bool;
         Spare10 : Bool;
         Spare9 : Bool;
         Spare8 : Bool;
         Spare7 : Bool;
         Spare6 : Bool;
         Spare5 : Bool;
         Spare4 : Bool;
         Spare3 : Bool;
         Spare2 : Bool;
         Spare1 : Bool;
      END_STRUCT;
      FP_EN : Struct
         Mode_Auto : Bool;
         Mode_Man : Bool;
         Mode_Loc : Bool;
         Mode_Test : Bool;
         Mode_SS_Field : Bool;
         Mode_SS_FP : Bool;
         PB_QStop : Bool;
         Spare9 : Bool;
         Spare8 : Bool;
         Spare7 : Bool;
         Spare6 : Bool;
         Spare5 : Bool;
         Spare4 : Bool;
         Spare3 : Bool;
         Spare2 : Bool;
         Spare1 : Bool;
      END_STRUCT;
      FP_DIM : Struct   // Faceplate Dimmed Buttons
         Auto : Bool;
         Local : Bool;
         Manual : Bool;
         Start1 : Bool;
         Start2 : Bool;
         Start3 : Bool;
         Stop : Bool;
         Test : Bool;
         QStop : Bool;
         Reset : Bool;
         Spare6 : Bool;
         Spare5 : Bool;
         Spare4 : Bool;
         Spare3 : Bool;
         Spare2 : Bool;
         Spare1 : Bool;
      END_STRUCT;
      FP_SHOW : Struct   // Faceplate Show Buttons
         PB_Auto : Bool;
         PB_Local : Bool;
         PB_Manual : Bool;
         PB_Start1 : Bool;
         PB_Start2 : Bool;
         PB_Start3 : Bool;
         PB_Stop : Bool;
         PB_Test : Bool;
         PB_QStop : Bool;
         AI1 : Bool;
         AI2 : Bool;
         AI3 : Bool;
         RDY : Bool;
         OVL : Bool;
         Spare1 : Bool;
         REM : Bool;
         SSW : Bool;
         DRDY : Bool;
         GFA : Bool;
         GWA : Bool;
         BUSF : Bool;
         Spare2 : Bool;
         UTEST : Bool;
         ACK : Bool;
         LSTR1 : Bool;
         LSTR2 : Bool;
         LSTR3 : Bool;
         INTL3 : Bool;
         CON3 : Bool;
         PREQ3 : Bool;
         LSP1 : Bool;
         LSP2 : Bool;
         LSP3 : Bool;
         RunTime : Bool;
         LimitDrift : Bool;
         PB_Reset : Bool;
         POS3 : Bool;
         Spare4 : Bool;
         Spare3 : Bool;
         Spare2_1 : Bool;
      END_STRUCT;
      FP_PARM : Struct   // Faceplate Parameters
         StartWarn_Pre : Int;
         StartWarn_Acc : Int;
         RunTime_Pre : Int;
         RunTime_Acc : Int;
         DriftingTime_Pre : Int;
         DriftingTime_Acc : Int;
         DelayStart_Pre : Int;
         DelayStart_Acc : Int;
         DelayStop_Pre : Int;
         DelayStop_Acc : Int;
         AI1_Max : Real;
         AI1_Min : Real;
         AI2_Max : Real;
         AI2_Min : Real;
         AI3_Max : Real;
         AI3_Min : Real;
         AO1a_Max : Real;
         AO1a_Min : Real;
         AO2a_Max : Real;
         AO2a_Min : Real;
         AO3a_Max : Real;
         AO3a_Min : Real;
         AO1b_Max : Real;
         AO1b_Min : Real;
         AO2b_Max : Real;
         AO2b_Min : Real;
         AO3b_Max : Real;
         AO3b_Min : Real;
         INTL : Bool;   // Interlock
         INTL_SEQ_STR1 : Bool;   // Interlock Sequence Start
         INTL_SEQ_STR2 : Bool;   // Interlock Sequence Start
         INTL_SEQ_STR3 : Bool;   // Interlock Sequence Start
         INTL_SEQ_STP : Bool;   // Interlock Sequence Stop
         T_Starting1 : Bool;
         T_Starting2 : Bool;
         T_Starting3 : Bool;
         Spare09 : Bool;
         Spare08 : Bool;
         Spare07 : Bool;
         Spare06 : Bool;
         Spare05 : Bool;
         Spare04 : Bool;
         Spare03 : Bool;
         Spare02 : Bool;
         Spare01 : Bool;
      END_STRUCT;
      FP_SIM : "ACESYS_SIM_VALVE";
      AdapterBlock : "ACESYS_ADPT_MOTOR";
      STATE : Struct
         A_Ctrl_AutoStart : Bool;
         A_Ctrl_DelayedStart1 : Bool;
         A_Ctrl_DelayedStart2 : Bool;
         A_Ctrl_DelayedStart3 : Bool;
         A_Ctrl_DelayedStop : Bool;
         A_Ctrl_MoveToPos1 : Bool;
         A_Ctrl_MoveToPos2 : Bool;
         A_Ctrl_MoveToPos3 : Bool;
         A_Ctrl_Parking1 : Bool;
         A_Ctrl_Parking2 : Bool;
         A_Ctrl_Parking3 : Bool;
         A_Ctrl_ParkStartWarning : Bool;
         A_Ctrl_Pos1 : Bool;
         A_Ctrl_Pos2 : Bool;
         A_Ctrl_Pos3 : Bool;
         A_Ctrl_Selected : Bool;
         A_Ctrl_SelToStop : Bool;
         A_Ctrl_SeqStart1 : Bool;
         A_Ctrl_SeqStart2 : Bool;
         A_Ctrl_SeqStart3 : Bool;
         A_Ctrl_SeqStop : Bool;
         A_Ctrl_StartWarning1 : Bool;
         A_Ctrl_StartWarning2 : Bool;
         A_Ctrl_StartWarning3 : Bool;
         A_Ctrl_Stopped : Bool;
         A_Ctrl_Stopping : Bool;
         A_NoCtrl_AutoStart : Bool;
         A_NoCtrl_Pos1 : Bool;
         A_NoCtrl_Pos2 : Bool;
         A_NoCtrl_Pos3 : Bool;
         A_NoCtrl_MoveToPos1 : Bool;
         A_NoCtrl_MoveToPos2 : Bool;
         A_NoCtrl_MoveToPos3 : Bool;
         A_NoCtrl_SeqStart1 : Bool;
         A_NoCtrl_SeqStart2 : Bool;
         A_NoCtrl_SeqStart3 : Bool;
         A_NoCtrl_StartWarning1 : Bool;
         A_NoCtrl_StartWarning2 : Bool;
         A_NoCtrl_StartWarning3 : Bool;
         S_AutoStart : Bool;
         S_MoveToPos1 : Bool;
         S_MoveToPos2 : Bool;
         S_MoveToPos3 : Bool;
         S_NotActive : Bool;
         S_Parking1 : Bool;
         S_Parking2 : Bool;
         S_Parking3 : Bool;
         S_ParkStartWarning : Bool;
         S_Pos1 : Bool;
         S_Pos2 : Bool;
         S_Pos3 : Bool;
         S_StartWarning1 : Bool;
         S_StartWarning2 : Bool;
         S_StartWarning3 : Bool;
         S_Stopping : Bool;
         M_AutoStart : Bool;
         M_MoveToPos1 : Bool;
         M_MoveToPos2 : Bool;
         M_MoveToPos3 : Bool;
         M_NotActive : Bool;
         M_Pos1 : Bool;
         M_Pos2 : Bool;
         M_Pos3 : Bool;
         M_StartWarning1 : Bool;
         M_StartWarning2 : Bool;
         M_StartWarning3 : Bool;
         L_AutoStart : Bool;
         L_MoveToPos1 : Bool;
         L_MoveToPos2 : Bool;
         L_MoveToPos3 : Bool;
         L_NotActive : Bool;
         L_Pos1 : Bool;
         L_Pos2 : Bool;
         L_Pos3 : Bool;
         L_StartWarning1 : Bool;
         L_StartWarning2 : Bool;
         L_StartWarning3 : Bool;
         T_TestMode : Bool;
         T_TestPermission : Bool;
         Alarm : Bool;
         Interlock : Bool;
         EmergencyStop : Bool;
         OutOfService : Bool;
      END_STRUCT;
      ONS : Struct
         Type_2Pos : Bool;
         Type_3Pos : Bool;
         Type_ConstantCmd : Bool;
         Type_PulseCmd : Bool;
         Type_NoLimit : Bool;
         LSP2_Off : Bool;
         LSTR1_2 : Bool;
         LSP3_On : Bool;
         LSTR2_2 : Bool;
         LSP3_Off : Bool;
         LSTR3_2 : Bool;
         AckAlarm_1 : Bool;
         AckAlarm : Bool;
         Cmd_Auto : Bool;
         Cmd_Manual : Bool;
         CMD_Local : Bool;
         CMD_Test : Bool;
         GLTP : Bool;
         MasterStop : Bool;
         LSP1_Off : Bool;
         LSP2_On : Bool;
         Park_Curr : Bool;
         Park_Pos1 : Bool;
         Park_Pos2 : Bool;
         Park_Pos3 : Bool;
         LSP1_On : Bool;
         CMD_Start1 : Bool;
         CMD_Start2 : Bool;
         CMD_Start3 : Bool;
         SecPulse1 : Bool;
         SecPulse2 : Bool;
         MovToPos : Bool;
      END_STRUCT;
      StatusWork : Int;
      ModePointer : Int;
      AlarmNo : Int;
      AlarmNo_Old : Int;
      StartWarn_Mem : Int;
      Runtime_Mem : Int;
      DriftingTime_Mem : Int;
      DelayStart_Mem : Int;
      DelayStop_Mem : Int;
      ModeAuto : Bool;
      ModeLocal : Bool;
      ModeManual : Bool;
      ModeSingleStart : Bool;
      ModeTest : Bool;
      Select : Bool;   // Parent & Program Select
      CMD_AckAlarm : Bool;
      CMD_Start1 : Bool;
      CMD_Start2 : Bool;
      CMD_Start3 : Bool;
      CMD_Stop : Bool;
      CMD_QStop : Bool;
      CMD_Reset : Bool;
      FromStateAuto : Bool;
      FromStateAuto_GrpCtrl : Bool;
      FromStateAuto_NoGrpCtrl : Bool;
      FromStateSingle : Bool;
      FromStateManual : Bool;
      FromStateLocal : Bool;
      FromStateTest : Bool;
      FromStopState : Bool;
      ALARM_SupressionActive : Bool;
      ALARM_AlarmPresent : Bool;
      ALARM_WarnPresent : Bool;
      ALARM_FailureAckRequired : Bool;
      ALARM_WarnAckRequired : Bool;
      StartWarn_TT : Bool;
      StartWarn_Done : Bool;
      RunTime_Done : Bool;
      DriftingTime_Done : Bool;
      DelayStart_Done : Bool;
      DelayStop_Done : Bool;
      Trig_ALARM_Runtime : Bool;
      Trig_ALARM_Drifting : Bool;
      LSTR1_Puls : Bool;
      LSTR2_Puls : Bool;
      LSTR3_Puls : Bool;
      DIR1_Request : Bool;
      DIR2_Request : Bool;
      DIR3_Request : Bool;
      LimitDrifting1 : Bool;
      LimitDrifting2 : Bool;
      LimitDrifting3 : Bool;
      LimitSwitchPos1Mem : Bool;
      LimitSwitchPos2Mem : Bool;
      LimitSwitchPos3Mem : Bool;
      CountElapsed_Wagging : Bool;
      Sec_Pulse : Bool;
      OUT : Struct
         CON1 : Bool;
         CON2 : Bool;
         CON3 : Bool;
         LAMP1 : Bool;
         LAMP2 : Bool;
         LAMP3 : Bool;
         SACK : Bool;
         POS1 : Bool;
         POS2 : Bool;
         POS3 : Bool;
         OK : Bool;
         LOC : Bool;
         MAN : Bool;
         AUT : Bool;
         SS : Bool;
         RES : Bool;
         TESTP : Bool;
         ASTW : Bool;
         AL_SUPR : Bool;
         INTL_OK_STAT : Bool;
         INTL_SEQ_STR1_OK_STAT : Bool;
         INTL_SEQ_STR2_OK_STAT : Bool;
         INTL_SEQ_STR3_OK_STAT : Bool;
         INTL_SEQ_STP_OK_STAT : Bool;
         MSW_EXT_ALARMFAILUNACK : Bool;
      END_STRUCT;
      MSW_Status_Trans : Int;
   END_VAR
   VAR_TEMP
      AOn : Bool;   // Always On
      AOff : Bool;   // Always Off
      DummyBool : Bool;
      StatPointer_Old : Int;
      StatusBuilder : Int;
      Status_Add : Int;
      LSP1_Temp : Bool;
      LSP2_Temp : Bool;
      LSP3_Temp : Bool;
      PREQ3_Temp : Bool;
   END_VAR
   VAR_TEMP   // added for the SCL form of the ladder/FBD networks
      _w1 : Bool;
      _w2 : Bool;
      _w3 : Bool;
      _w4 : Bool;
      _w5 : Bool;
      _w6 : Bool;
   END_VAR
BEGIN

REGION Network 1: Always On
